C09130=1221.098,210.691,-57.647,-177.348,6.190,148.329
C09131=1221.102,210.442,-57.622,-177.351,6.188,148.329
C09132=1221.107,210.193,-57.597,-177.354,6.186,148.330
C09133=1221.111,209.944,-57.573,-177.356,6.184,148.330
C09134=1221.117,209.695,-57.549,-177.359,6.183,148.330
C09135=1221.121,209.446,-57.525,-177.361,6.181,148.331
C09136=1221.125,209.197,-57.501,-177.364,6.179,148.331
C09137=1221.130,208.949,-57.476,-177.367,6.177,148.331
C09138=1221.134,208.700,-57.452,-177.369,6.176,148.332
C09139=1221.138,208.451,-57.428,-177.371,6.174,148.332
C09140=1221.144,208.202,-57.404,-177.374,6.172,148.332
C09141=1221.148,207.953,-57.380,-177.377,6.171,148.333
C09142=1221.153,207.705,-57.356,-177.380,6.169,148.333
C09143=1221.158,207.456,-57.331,-177.382,6.167,148.334
C09144=1221.161,207.207,-57.307,-177.385,6.165,148.334
C09145=1221.166,206.958,-57.283,-177.388,6.163,148.334
C09146=1221.171,206.710,-57.259,-177.390,6.162,148.335
C09147=1221.176,206.461,-57.234,-177.392,6.161,148.335
C09148=1221.180,206.212,-57.211,-177.395,6.159,148.335
C09149=1221.185,205.964,-57.187,-177.398,6.157,148.336
C09150=1221.189,205.715,-57.163,-177.400,6.155,148.336
C09151=1221.194,205.466,-57.138,-177.403,6.153,148.336
C09152=1221.198,205.217,-57.115,-177.406,6.151,148.337
C09153=1221.203,204.968,-57.090,-177.408,6.150,148.337
C09154=1221.207,204.720,-57.066,-177.410,6.148,148.337
C09155=1221.213,204.471,-57.042,-177.413,6.147,148.338
C09156=1221.216,204.221,-57.018,-177.416,6.145,148.338
C09157=1221.221,203.973,-56.994,-177.418,6.143,148.338
C09158=1221.225,203.724,-56.971,-177.421,6.141,148.339
C09159=1221.230,203.476,-56.946,-177.424,6.139,148.339
C09160=1221.235,203.226,-56.923,-177.426,6.138,148.339
C09161=1221.240,202.978,-56.898,-177.428,6.136,148.340
C09162=1221.244,202.729,-56.875,-177.431,6.135,148.340
C09163=1221.248,202.480,-56.851,-177.434,6.133,148.340
C09164=1221.253,202.231,-56.827,-177.436,6.131,148.341
C09165=1221.257,201.982,-56.803,-177.439,6.129,148.341
C09166=1221.262,201.734,-56.779,-177.441,6.128,148.342
C09167=1221.267,201.485,-56.755,-177.444,6.126,148.342
C09168=1221.272,201.236,-56.731,-177.447,6.125,148.342
C09169=1221.276,200.987,-56.708,-177.449,6.123,148.343
C09170=1221.281,200.739,-56.684,-177.452,6.121,148.343
C09171=1221.285,200.490,-56.660,-177.454,6.120,148.344
C09172=1221.290,200.241,-56.636,-177.457,6.118,148.344
C09173=1221.294,199.992,-56.613,-177.459,6.116,148.344
C09174=1221.298,199.743,-56.588,-177.462,6.114,148.345
C09175=1221.303,199.494,-56.565,-177.465,6.113,148.345
C09176=1221.308,199.245,-56.542,-177.467,6.111,148.345
C09177=1221.312,198.997,-56.518,-177.469,6.110,148.346
C09178=1221.317,198.747,-56.494,-177.472,6.108,148.346
C09179=1221.322,198.499,-56.470,-177.475,6.106,148.347
C09180=1221.327,198.250,-56.446,-177.478,6.104,148.347
C09181=1221.331,198.001,-56.423,-177.480,6.103,148.347
C09182=1221.336,197.752,-56.399,-177.482,6.102,148.348
C09183=1221.340,197.503,-56.375,-177.485,6.100,148.348
C09184=1221.345,197.254,-56.352,-177.488,6.098,148.348
C09185=1221.349,197.006,-56.328,-177.490,6.096,148.349
C09186=1221.354,196.757,-56.305,-177.493,6.094,148.349
C09187=1221.359,196.508,-56.281,-177.495,6.093,148.349
C09188=1221.363,196.259,-56.257,-177.498,6.091,148.350
C09189=1221.368,196.010,-56.234,-177.500,6.090,148.350
C09190=1221.373,195.761,-56.211,-177.504,6.088,148.351
C09191=1221.377,195.512,-56.187,-177.506,6.086,148.351
C09192=1221.382,195.264,-56.163,-177.508,6.085,148.351
C09193=1221.386,195.015,-56.140,-177.511,6.083,148.352
C09194=1221.390,194.766,-56.117,-177.514,6.082,148.352
C09195=1221.395,194.517,-56.094,-177.516,6.080,148.352
C09196=1221.399,194.269,-56.070,-177.519,6.078,148.353
C09197=1221.404,194.020,-56.046,-177.521,6.077,148.353
C09198=1221.409,193.771,-56.023,-177.524,6.075,148.353
C09199=1221.414,193.522,-55.999,-177.526,6.073,148.354
C09200=1221.418,193.273,-55.976,-177.529,6.072,148.354
C09201=1221.423,193.024,-55.952,-177.531,6.071,148.355
C09202=1221.427,192.775,-55.929,-177.534,6.069,148.355
C09203=1221.433,192.527,-55.906,-177.537,6.067,148.355
C09204=1221.437,192.278,-55.883,-177.539,6.065,148.356
C09205=1221.441,192.029,-55.860,-177.541,6.064,148.356
C09206=1221.446,191.780,-55.836,-177.544,6.062,148.356
C09207=1221.451,191.531,-55.813,-177.547,6.060,148.357
C09208=1221.455,191.282,-55.789,-177.550,6.059,148.357
C09209=1221.460,191.033,-55.766,-177.553,6.057,148.358
C09210=1221.465,190.784,-55.743,-177.555,6.056,148.358
C09211=1221.468,190.536,-55.719,-177.557,6.054,148.358
C09212=1221.473,190.287,-55.696,-177.560,6.052,148.359
C09213=1221.478,190.038,-55.673,-177.563,6.051,148.359
C09214=1221.483,189.789,-55.650,-177.565,6.050,148.360
C09215=1221.488,189.540,-55.626,-177.567,6.048,148.360
C09216=1221.492,189.292,-55.603,-177.570,6.046,148.360
C09217=1221.497,189.043,-55.580,-177.573,6.044,148.361
C09218=1221.501,188.794,-55.557,-177.575,6.043,148.361
C09219=1221.506,188.545,-55.533,-177.578,6.042,148.362
C09220=1221.510,188.296,-55.511,-177.580,6.040,148.362
C09221=1221.515,188.047,-55.487,-177.583,6.038,148.362
C09222=1221.520,187.798,-55.465,-177.586,6.037,148.363
C09223=1221.525,187.549,-55.442,-177.588,6.035,148.363
C09224=1221.529,187.300,-55.419,-177.591,6.034,148.364
C09225=1221.534,187.051,-55.395,-177.593,6.033,148.364
C09226=1221.538,186.802,-55.372,-177.596,6.031,148.364
C09227=1221.543,186.553,-55.349,-177.598,6.029,148.365
C09228=1221.548,186.305,-55.326,-177.601,6.027,148.365
C09229=1221.552,186.056,-55.303,-177.604,6.026,148.366
C09230=1221.558,185.786,-55.278,-177.606,6.024,148.366
C09231=1221.562,185.517,-55.254,-177.609,6.023,148.366
C09232=1221.567,185.247,-55.229,-177.612,6.021,148.367
C09233=1221.572,184.977,-55.204,-177.615,6.019,148.367
C09234=1221.577,184.728,-55.181,-177.617,6.017,148.368
C09235=1221.581,184.479,-55.157,-177.620,6.016,148.368
C09236=1221.586,184.230,-55.135,-177.622,6.015,148.368
C09237=1221.590,183.981,-55.112,-177.625,6.013,148.369
C09238=1221.596,183.733,-55.089,-177.628,6.011,148.369
C09239=1221.600,183.484,-55.066,-177.631,6.009,148.370
C09240=1221.604,183.235,-55.043,-177.633,6.008,148.370
C09241=1221.609,182.985,-55.020,-177.635,6.007,148.370
C09242=1221.613,182.737,-54.997,-177.638,6.005,148.371
C09243=1221.619,182.488,-54.974,-177.640,6.004,148.371
C09244=1221.623,182.239,-54.952,-177.643,6.002,148.372
C09245=1221.628,181.990,-54.929,-177.646,6.000,148.372
C09246=1221.632,181.741,-54.906,-177.648,5.999,148.372
C09247=1221.637,181.493,-54.883,-177.651,5.998,148.373
C09248=1221.642,181.243,-54.861,-177.654,5.996,148.373
C09249=1221.646,180.994,-54.838,-177.656,5.994,148.374
C09250=1221.651,180.745,-54.815,-177.658,5.993,148.374
C09251=1221.655,180.497,-54.793,-177.661,5.991,148.374
C09252=1221.660,180.248,-54.769,-177.664,5.990,148.375
C09253=1221.664,179.998,-54.747,-177.666,5.989,148.375
C09254=1221.670,179.750,-54.724,-177.669,5.987,148.376
C09255=1221.674,179.501,-54.702,-177.672,5.985,148.376
C09256=1221.679,179.252,-54.679,-177.674,5.984,148.376
C09257=1221.683,179.003,-54.656,-177.676,5.982,148.377
C09258=1221.688,178.754,-54.634,-177.679,5.981,148.377
C09259=1221.692,178.505,-54.611,-177.682,5.980,148.378
C09260=1221.697,178.256,-54.589,-177.684,5.978,148.378
C09261=1221.702,178.008,-54.566,-177.687,5.976,148.378
C09262=1221.706,177.759,-54.543,-177.689,5.975,148.379
C09263=1221.711,177.509,-54.521,-177.692,5.974,148.379
C09264=1221.715,177.261,-54.498,-177.695,5.972,148.380
C09265=1221.720,177.012,-54.476,-177.697,5.971,148.380
C09266=1221.724,176.763,-54.453,-177.699,5.969,148.381
C09267=1221.730,176.514,-54.431,-177.703,5.968,148.381
C09268=1221.734,176.265,-54.409,-177.705,5.967,148.381
C09269=1221.739,176.016,-54.385,-177.707,5.965,148.382
C09270=1221.744,175.767,-54.364,-177.710,5.963,148.382
C09271=1221.748,175.518,-54.341,-177.712,5.962,148.383
C09272=1221.753,175.269,-54.318,-177.715,5.961,148.383
C09273=1221.757,175.021,-54.296,-177.718,5.959,148.384
C09274=1221.762,174.771,-54.273,-177.720,5.958,148.384
C09275=1221.767,174.522,-54.251,-177.723,5.956,148.384
C09276=1221.771,174.274,-54.229,-177.726,5.954,148.385
C09277=1221.776,174.024,-54.206,-177.728,5.953,148.385
C09278=1221.781,173.776,-54.184,-177.731,5.952,148.386
C09279=1221.785,173.526,-54.162,-177.733,5.950,148.386
C09280=1221.790,173.277,-54.139,-177.736,5.949,148.387
C09281=1221.794,173.029,-54.117,-177.738,5.947,148.387
C09282=1221.799,172.779,-54.095,-177.741,5.945,148.387
C09283=1221.804,172.531,-54.072,-177.743,5.944,148.388
C09284=1221.809,172.281,-54.050,-177.746,5.943,148.388
C09285=1221.813,172.033,-54.028,-177.748,5.942,148.389
C09286=1221.818,171.784,-54.005,-177.751,5.940,148.389
C09287=1221.822,171.534,-53.983,-177.754,5.938,148.389
C09288=1221.827,171.286,-53.961,-177.756,5.938,148.390
C09289=1221.831,171.037,-53.939,-177.759,5.936,148.390
C09290=1221.837,170.788,-53.916,-177.762,5.934,148.391
C09291=1221.841,170.539,-53.894,-177.764,5.933,148.391
C09292=1221.846,170.291,-53.872,-177.767,5.931,148.392
C09293=1221.851,170.041,-53.849,-177.770,5.930,148.392
C09294=1221.856,169.792,-53.828,-177.772,5.929,148.392
C09295=1221.860,169.543,-53.806,-177.774,5.927,148.393
C09296=1221.864,169.294,-53.784,-177.777,5.926,148.393
C09297=1221.869,169.045,-53.762,-177.780,5.924,148.394
C09298=1221.874,168.796,-53.738,-177.782,5.923,148.394
C09299=1221.879,168.547,-53.717,-177.784,5.922,148.394
C09300=1221.883,168.298,-53.695,-177.787,5.920,148.395
C09301=1221.888,168.049,-53.673,-177.790,5.919,148.395
C09302=1221.893,167.800,-53.650,-177.792,5.917,148.396
C09303=1221.898,167.551,-53.629,-177.795,5.915,148.396
C09304=1221.902,167.302,-53.607,-177.797,5.915,148.397
C09305=1221.907,167.053,-53.585,-177.800,5.913,148.397
C09306=1221.911,166.804,-53.562,-177.803,5.911,148.398
C09307=1221.916,166.556,-53.541,-177.805,5.910,148.398
C09308=1221.920,166.306,-53.518,-177.808,5.909,148.399
C09309=1221.925,166.057,-53.496,-177.810,5.908,148.399
C09310=1221.930,165.808,-53.474,-177.813,5.906,148.399
C09311=1221.935,165.559,-53.452,-177.815,5.905,148.400
C09312=1221.939,165.310,-53.430,-177.818,5.903,148.400
C09313=1221.944,165.061,-53.409,-177.821,5.901,148.401
C09314=1221.949,164.813,-53.387,-177.823,5.901,148.401
C09315=1221.953,164.563,-53.365,-177.826,5.899,148.402
C09316=1221.958,164.315,-53.343,-177.828,5.898,148.402
C09317=1221.962,164.065,-53.321,-177.831,5.896,148.402
C09318=1221.968,163.816,-53.299,-177.834,5.895,148.403
C09319=1221.972,163.567,-53.277,-177.836,5.894,148.403
C09320=1221.977,163.318,-53.255,-177.839,5.892,148.404
C09321=1221.981,163.069,-53.233,-177.841,5.891,148.404
C09322=1221.986,162.820,-53.212,-177.844,5.889,148.405
C09323=1221.991,162.571,-53.191,-177.847,5.888,148.405
C09324=1221.995,162.322,-53.169,-177.849,5.887,148.406
C09325=1222.000,162.073,-53.147,-177.852,5.885,148.406
C09326=1222.004,161.824,-53.125,-177.854,5.884,148.406
C09327=1222.009,161.575,-53.103,-177.857,5.883,148.407
C09328=1222.014,161.327,-53.081,-177.859,5.882,148.407
C09329=1222.018,161.077,-53.059,-177.862,5.880,148.408
C09330=1222.024,160.828,-53.038,-177.864,5.878,148.408
C09331=1222.028,160.579,-53.016,-177.867,5.877,148.409
C09332=1222.033,160.330,-52.995,-177.870,5.876,148.409
C09333=1222.038,160.081,-52.973,-177.872,5.875,148.410
C09334=1222.042,159.812,-52.950,-177.875,5.873,148.410
C09335=1222.048,159.544,-52.926,-177.878,5.871,148.410
C09336=1222.052,159.274,-52.902,-177.881,5.870,148.411
C09337=1222.057,159.004,-52.880,-177.883,5.869,148.411
C09338=1222.062,158.756,-52.858,-177.886,5.867,148.412
C09339=1222.067,158.507,-52.836,-177.888,5.866,148.412
C09340=1222.071,158.257,-52.815,-177.891,5.865,148.413
C09341=1222.076,158.009,-52.793,-177.893,5.864,148.413
C09342=1222.081,157.760,-52.772,-177.896,5.862,148.414
C09343=1222.085,157.511,-52.750,-177.899,5.860,148.414
C09344=1222.091,157.261,-52.729,-177.901,5.860,148.415
C09345=1222.096,157.013,-52.707,-177.904,5.858,148.415
C09346=1222.099,156.764,-52.685,-177.906,5.857,148.416
C09347=1222.104,156.514,-52.665,-177.909,5.855,148.416
C09348=1222.109,156.266,-52.643,-177.911,5.854,148.417
C09349=1222.113,156.016,-52.621,-177.914,5.853,148.417
C09350=1222.119,155.767,-52.600,-177.917,5.852,148.418
C09351=1222.123,155.519,-52.578,-177.919,5.850,148.418
C09352=1222.128,155.270,-52.556,-177.922,5.849,148.419
C09353=1222.133,155.020,-52.535,-177.924,5.848,148.419
C09354=1222.137,154.772,-52.514,-177.927,5.847,148.419
C09355=1222.142,154.522,-52.493,-177.930,5.845,148.420
C09356=1222.146,154.273,-52.471,-177.932,5.843,148.420
C09357=1222.152,154.024,-52.450,-177.934,5.842,148.421
C09358=1222.156,153.775,-52.428,-177.938,5.841,148.421
C09359=1222.161,153.527,-52.407,-177.940,5.840,148.422
C09360=1222.165,153.277,-52.386,-177.942,5.838,148.422
C09361=1222.170,153.028,-52.364,-177.945,5.837,148.423
C09362=1222.175,152.779,-52.343,-177.948,5.836,148.423
C09363=1222.180,152.530,-52.322,-177.950,5.835,148.423
C09364=1222.184,152.281,-52.301,-177.953,5.833,148.424
C09365=1222.189,152.032,-52.279,-177.955,5.832,148.424
C09366=1222.194,151.783,-52.258,-177.958,5.831,148.425
C09367=1222.199,151.534,-52.237,-177.960,5.830,148.425
C09368=1222.203,151.285,-52.216,-177.963,5.828,148.426
C09369=1222.208,151.036,-52.194,-177.966,5.827,148.426
C09370=1222.213,150.787,-52.173,-177.968,5.825,148.427
C09371=1222.218,150.537,-52.152,-177.970,5.824,148.427
C09372=1222.222,150.289,-52.131,-177.973,5.823,148.428
C09373=1222.227,150.039,-52.110,-177.976,5.822,148.428
C09374=1222.231,149.790,-52.088,-177.979,5.820,148.429
C09375=1222.236,149.541,-52.068,-177.981,5.820,148.429
C09376=1222.241,149.292,-52.047,-177.984,5.818,148.430
C09377=1222.246,149.044,-52.025,-177.986,5.817,148.430
C09378=1222.250,148.794,-52.004,-177.989,5.815,148.431
C09379=1222.255,148.545,-51.983,-177.991,5.814,148.431
C09380=1222.260,148.296,-51.962,-177.994,5.813,148.432
C09381=1222.264,148.047,-51.941,-177.996,5.812,148.432
C09382=1222.269,147.798,-51.920,-177.999,5.810,148.433
C09383=1222.274,147.549,-51.899,-178.001,5.809,148.433
C09384=1222.278,147.299,-51.878,-178.004,5.808,148.433
C09385=1222.283,147.050,-51.857,-178.007,5.807,148.434
C09386=1222.288,146.802,-51.835,-178.009,5.805,148.434
C09387=1222.293,146.553,-51.815,-178.012,5.804,148.435
C09388=1222.298,146.303,-51.794,-178.015,5.803,148.435
C09389=1222.302,146.054,-51.774,-178.017,5.802,148.436
C09390=1222.307,145.806,-51.752,-178.019,5.801,148.436
C09391=1222.312,145.556,-51.731,-178.022,5.799,148.437
C09392=1222.316,145.307,-51.710,-178.025,5.799,148.437
C09393=1222.321,145.058,-51.689,-178.027,5.797,148.438
C09394=1222.325,144.809,-51.668,-178.029,5.796,148.438
C09395=1222.331,144.560,-51.647,-178.033,5.794,148.439
C09396=1222.335,144.311,-51.627,-178.035,5.793,148.439
C09397=1222.340,144.062,-51.606,-178.038,5.792,148.440
C09398=1222.345,143.813,-51.585,-178.040,5.791,148.440
C09399=1222.349,143.563,-51.564,-178.043,5.789,148.441
C09400=1222.354,143.314,-51.542,-178.045,5.788,148.441
C09401=1222.359,143.065,-51.522,-178.048,5.787,148.441
C09402=1222.364,142.816,-51.501,-178.050,5.786,148.442
C09403=1222.368,142.567,-51.481,-178.053,5.785,148.443
C09404=1222.373,142.318,-51.460,-178.056,5.784,148.443
C09405=1222.378,142.069,-51.439,-178.058,5.783,148.444
C09406=1222.383,141.820,-51.418,-178.061,5.781,148.444
C09407=1222.387,141.571,-51.398,-178.063,5.780,148.445
C09408=1222.392,141.322,-51.378,-178.066,5.778,148.445
C09409=1222.397,141.073,-51.356,-178.068,5.778,148.446
C09410=1222.401,140.824,-51.336,-178.071,5.776,148.446
C09411=1222.406,140.575,-51.315,-178.074,5.775,148.447
C09412=1222.411,140.326,-51.294,-178.076,5.774,148.447
C09413=1222.416,140.077,-51.273,-178.079,5.773,148.448
C09414=1222.420,139.827,-51.253,-178.081,5.772,148.448
C09415=1222.425,139.578,-51.232,-178.084,5.770,148.448
C09416=1222.429,139.329,-51.211,-178.086,5.769,148.449
C09417=1222.434,139.080,-51.191,-178.089,5.768,148.449
C09418=1222.439,138.831,-51.170,-178.092,5.767,148.450
C09419=1222.443,138.582,-51.150,-178.094,5.765,148.450
C09420=1222.449,138.332,-51.129,-178.097,5.764,148.451
C09421=1222.453,138.083,-51.108,-178.099,5.764,148.451
C09422=1222.458,137.834,-51.089,-178.102,5.762,148.452
C09423=1222.463,137.585,-51.068,-178.104,5.761,148.452
C09424=1222.467,137.336,-51.047,-178.107,5.759,148.453
C09425=1222.473,137.086,-51.026,-178.109,5.759,148.453
C09426=1222.477,136.837,-51.006,-178.112,5.758,148.454
C09427=1222.481,136.588,-50.985,-178.115,5.756,148.454
C09428=1222.487,136.339,-50.965,-178.117,5.755,148.455
C09429=1222.491,136.090,-50.944,-178.120,5.754,148.455
C09430=1222.495,135.841,-50.924,-178.122,5.753,148.456
C09431=1222.502,135.592,-50.904,-178.125,5.751,148.456
C09432=1222.506,135.343,-50.884,-178.127,5.750,148.457
C09433=1222.510,135.094,-50.863,-178.130,5.750,148.457
C09434=1222.516,134.845,-50.842,-178.133,5.748,148.458
C09435=1222.520,134.596,-50.822,-178.135,5.747,148.459
C09436=1222.524,134.347,-50.801,-178.138,5.745,148.459
C09437=1222.529,134.098,-50.782,-178.140,5.745,148.459
C09438=1222.535,133.829,-50.759,-178.143,5.743,148.460
C09439=1222.540,133.560,-50.737,-178.146,5.742,148.461
C09440=1222.544,133.291,-50.716,-178.149,5.741,148.461
C09441=1222.550,133.023,-50.694,-178.151,5.740,148.462
C09442=1222.554,132.774,-50.673,-178.154,5.739,148.462
C09443=1222.559,132.524,-50.653,-178.156,5.738,148.463
C09444=1222.564,132.275,-50.632,-178.159,5.737,148.463
C09445=1222.569,132.026,-50.612,-178.162,5.735,148.464
C09446=1222.574,131.778,-50.592,-178.164,5.734,148.464
C09447=1222.578,131.529,-50.572,-178.167,5.733,148.465
C09448=1222.584,131.279,-50.552,-178.170,5.732,148.465
C09449=1222.588,131.030,-50.531,-178.172,5.731,148.466
C09450=1222.592,130.781,-50.511,-178.174,5.729,148.466
C09451=1222.597,130.531,-50.491,-178.177,5.729,148.467
C09452=1222.602,130.282,-50.471,-178.180,5.727,148.467
C09453=1222.607,130.033,-50.450,-178.182,5.726,148.468
C09454=1222.612,129.783,-50.430,-178.184,5.725,148.468
C09455=1222.617,129.535,-50.410,-178.188,5.724,148.469
C09456=1222.621,129.286,-50.390,-178.190,5.723,148.469
C09457=1222.626,129.037,-50.370,-178.192,5.722,148.470
C09458=1222.630,128.788,-50.350,-178.195,5.720,148.470
C09459=1222.636,128.538,-50.330,-178.198,5.720,148.471
C09460=1222.640,128.289,-50.309,-178.200,5.718,148.471
C09461=1222.645,128.040,-50.289,-178.203,5.717,148.472
C09462=1222.650,127.791,-50.270,-178.205,5.716,148.472
C09463=1222.654,127.542,-50.249,-178.208,5.715,148.473
C09464=1222.659,127.293,-50.230,-178.210,5.714,148.473
C09465=1222.664,127.044,-50.209,-178.213,5.713,148.474
C09466=1222.668,126.794,-50.190,-178.216,5.712,148.474
C09467=1222.673,126.546,-50.170,-178.218,5.711,148.475
C09468=1222.679,126.296,-50.149,-178.221,5.710,148.476
C09469=1222.683,126.047,-50.129,-178.223,5.708,148.476
C09470=1222.688,125.797,-50.109,-178.226,5.708,148.477
C09471=1222.692,125.549,-50.089,-178.229,5.706,148.477
C09472=1222.697,125.299,-50.069,-178.231,5.705,148.478
C09473=1222.702,125.051,-50.049,-178.233,5.704,148.478
C09474=1222.707,124.801,-50.030,-178.237,5.703,148.479
C09475=1222.712,124.552,-50.010,-178.239,5.702,148.479
C09476=1222.716,124.303,-49.990,-178.241,5.701,148.480
C09477=1222.721,124.054,-49.970,-178.244,5.700,148.480
C09478=1222.726,123.805,-49.950,-178.247,5.699,148.481
C09479=1222.731,123.555,-49.930,-178.249,5.698,148.481
C09480=1222.735,123.306,-49.911,-178.252,5.697,148.482
C09481=1222.740,123.057,-49.890,-178.254,5.696,148.482
C09482=1222.745,122.808,-49.871,-178.257,5.695,148.483
C09483=1222.750,122.558,-49.851,-178.259,5.693,148.483
C09484=1222.754,122.309,-49.831,-178.262,5.693,148.484
C09485=1222.759,122.060,-49.811,-178.264,5.692,148.484
C09486=1222.764,121.812,-49.791,-178.267,5.690,148.485
C09487=1222.769,121.562,-49.772,-178.270,5.690,148.485
C09488=1222.774,121.312,-49.752,-178.272,5.689,148.486
C09489=1222.779,121.064,-49.733,-178.275,5.687,148.486
C09490=1222.783,120.815,-49.712,-178.277,5.686,148.487
C09491=1222.788,120.565,-49.693,-178.280,5.686,148.487
C09492=1222.792,120.316,-49.674,-178.282,5.684,148.488
C09493=1222.797,120.067,-49.654,-178.285,5.683,148.489
C09494=1222.802,119.818,-49.634,-178.287,5.682,148.489
C09495=1222.807,119.568,-49.614,-178.290,5.681,148.490
C09496=1222.812,119.319,-49.595,-178.292,5.680,148.490
C09497=1222.817,119.070,-49.575,-178.295,5.679,148.491
C09498=1222.821,118.821,-49.555,-178.298,5.679,148.491
C09499=1222.827,118.572,-49.536,-178.300,5.677,148.492
C09500=1222.831,118.323,-49.516,-178.303,5.676,148.492
C09501=1222.836,118.073,-49.496,-178.305,5.675,148.493
C09502=1222.841,117.824,-49.478,-178.308,5.674,148.493
C09503=1222.845,117.575,-49.457,-178.310,5.673,148.494
C09504=1222.850,117.326,-49.438,-178.313,5.672,148.494
C09505=1222.855,117.077,-49.418,-178.316,5.671,148.495
C09506=1222.860,116.827,-49.399,-178.318,5.670,148.495
C09507=1222.865,116.578,-49.379,-178.321,5.669,148.496
C09508=1222.869,116.329,-49.360,-178.324,5.667,148.496
C09509=1222.874,116.080,-49.341,-178.326,5.667,148.497
C09510=1222.878,115.831,-49.320,-178.328,5.666,148.497
C09511=1222.884,115.582,-49.301,-178.331,5.665,148.498
C09512=1222.889,115.332,-49.281,-178.334,5.663,148.499
C09513=1222.893,115.083,-49.262,-178.336,5.663,148.499
C09514=1222.898,114.834,-49.243,-178.339,5.662,148.500
C09515=1222.903,114.585,-49.223,-178.342,5.660,148.500
C09516=1222.908,114.336,-49.204,-178.344,5.660,148.501
C09517=1222.913,114.086,-49.184,-178.346,5.659,148.501
C09518=1222.917,113.837,-49.165,-178.349,5.658,148.502
C09519=1222.922,113.588,-49.146,-178.352,5.657,148.503
C09520=1222.927,113.339,-49.126,-178.354,5.656,148.503
C09521=1222.932,113.090,-49.107,-178.357,5.655,148.504
C09522=1222.936,112.840,-49.088,-178.359,5.653,148.504
C09523=1222.941,112.591,-49.068,-178.362,5.653,148.505
C09524=1222.946,112.342,-49.049,-178.364,5.652,148.505
C09525=1222.951,112.092,-49.030,-178.367,5.651,148.506
C09526=1222.956,111.844,-49.011,-178.370,5.650,148.506
C09527=1222.960,111.594,-48.991,-178.372,5.649,148.507
C09528=1222.966,111.345,-48.972,-178.375,5.648,148.507
C09529=1222.970,111.096,-48.953,-178.377,5.647,148.508
C09530=1222.974,110.847,-48.933,-178.380,5.646,148.508
C09531=1222.980,110.598,-48.914,-178.383,5.645,148.509
C09532=1222.984,110.348,-48.896,-178.385,5.644,148.509
C09533=1222.989,110.099,-48.876,-178.387,5.644,148.510
C09534=1222.994,109.849,-48.857,-178.390,5.642,148.510
C09535=1222.999,109.601,-48.838,-178.393,5.641,148.511
C09536=1223.004,109.351,-48.818,-178.395,5.640,148.512
C09537=1223.009,109.102,-48.799,-178.398,5.639,148.512
C09538=1223.013,108.853,-48.780,-178.401,5.638,148.513
C09539=1223.019,108.604,-48.761,-178.403,5.637,148.513
C09540=1223.023,108.354,-48.742,-178.405,5.637,148.514
C09541=1223.028,108.106,-48.723,-178.409,5.635,148.514
C09542=1223.033,107.837,-48.702,-178.411,5.634,148.515
C09543=1223.038,107.568,-48.681,-178.413,5.634,148.516
C09544=1223.044,107.300,-48.661,-178.416,5.632,148.516
C09545=1223.048,107.031,-48.640,-178.419,5.631,148.517
C09546=1223.053,106.783,-48.621,-178.422,5.631,148.517
C09547=1223.059,106.533,-48.602,-178.424,5.629,148.518
C09548=1223.063,106.284,-48.583,-178.427,5.628,148.519
C09549=1223.068,106.035,-48.564,-178.429,5.628,148.519
C09550=1223.072,105.786,-48.545,-178.432,5.627,148.520
C09551=1223.078,105.536,-48.526,-178.435,5.625,148.520
C09552=1223.082,105.287,-48.507,-178.437,5.625,148.521
C09553=1223.087,105.038,-48.488,-178.440,5.624,148.521
C09554=1223.091,104.788,-48.470,-178.442,5.623,148.522
C09555=1223.097,104.539,-48.450,-178.445,5.622,148.522
C09556=1223.101,104.290,-48.431,-178.448,5.621,148.523
C09557=1223.106,104.041,-48.413,-178.450,5.620,148.523
C09558=1223.111,103.791,-48.393,-178.452,5.619,148.524
C09559=1223.116,103.542,-48.374,-178.455,5.618,148.525
C09560=1223.121,103.293,-48.356,-178.458,5.617,148.525
C09561=1223.125,103.044,-48.337,-178.460,5.616,148.526
C09562=1223.131,102.795,-48.318,-178.463,5.616,148.526
C09563=1223.135,102.545,-48.299,-178.465,5.615,148.527
C09564=1223.140,102.296,-48.280,-178.468,5.613,148.527
C09565=1223.145,102.046,-48.262,-178.471,5.613,148.528
C09566=1223.149,101.798,-48.243,-178.473,5.612,148.528
C09567=1223.155,101.549,-48.224,-178.475,5.611,148.529
C09568=1223.159,101.299,-48.205,-178.478,5.609,148.530
C09569=1223.164,101.050,-48.186,-178.481,5.609,148.530
C09570=1223.169,100.800,-48.168,-178.483,5.608,148.531
C09571=1223.174,100.551,-48.148,-178.486,5.607,148.531
C09572=1223.179,100.302,-48.130,-178.488,5.607,148.532
C09573=1223.183,100.053,-48.111,-178.491,5.605,148.533
C09574=1223.188,99.803,-48.093,-178.493,5.604,148.533
C09575=1223.192,99.554,-48.074,-178.496,5.604,148.534
C09576=1223.198,99.305,-48.055,-178.499,5.603,148.534
C09577=1223.203,99.056,-48.036,-178.501,5.602,148.535
C09578=1223.207,98.806,-48.018,-178.504,5.601,148.535
C09579=1223.212,98.557,-47.999,-178.507,5.600,148.536
C09580=1223.217,98.308,-47.981,-178.509,5.599,148.536
C09581=1223.221,98.059,-47.962,-178.511,5.599,148.537
C09582=1223.227,97.809,-47.943,-178.514,5.598,148.538
C09583=1223.232,97.561,-47.924,-178.517,5.596,148.538
C09584=1223.237,97.311,-47.905,-178.519,5.596,148.539
C09585=1223.242,97.061,-47.887,-178.522,5.595,148.539
C09586=1223.246,96.813,-47.869,-178.524,5.594,148.540
C09587=1223.251,96.563,-47.850,-178.527,5.593,148.540
C09588=1223.256,96.314,-47.831,-178.529,5.593,148.541
C09589=1223.261,96.065,-47.813,-178.532,5.591,148.541
C09590=1223.265,95.815,-47.795,-178.535,5.590,148.542
C09591=1223.270,95.566,-47.776,-178.537,5.590,148.543
C09592=1223.275,95.317,-47.758,-178.539,5.589,148.543
C09593=1223.280,95.067,-47.739,-178.542,5.588,148.544
C09594=1223.285,94.818,-47.720,-178.545,5.587,148.544
C09595=1223.290,94.569,-47.702,-178.547,5.586,148.545
C09596=1223.294,94.319,-47.684,-178.550,5.585,148.546
C09597=1223.299,94.071,-47.665,-178.553,5.585,148.546
C09598=1223.304,93.821,-47.646,-178.555,5.584,148.547
C09599=1223.309,93.572,-47.628,-178.557,5.583,148.547
C09600=1223.313,93.323,-47.609,-178.560,5.582,148.548
C09601=1223.318,93.074,-47.591,-178.563,5.581,148.548
C09602=1223.324,92.824,-47.573,-178.565,5.580,148.549
C09603=1223.328,92.574,-47.554,-178.568,5.580,148.550
C09604=1223.333,92.326,-47.536,-178.570,5.579,148.550
C09605=1223.338,92.077,-47.518,-178.573,5.578,148.551
C09606=1223.343,91.827,-47.499,-178.576,5.577,148.551
C09607=1223.348,91.577,-47.481,-178.578,5.576,148.552
C09608=1223.352,91.329,-47.462,-178.581,5.575,148.552
C09609=1223.357,91.079,-47.444,-178.583,5.574,148.553
C09610=1223.362,90.830,-47.426,-178.586,5.574,148.554
C09611=1223.366,90.580,-47.408,-178.588,5.573,148.554
C09612=1223.372,90.331,-47.389,-178.591,5.571,148.555
C09613=1223.377,90.082,-47.371,-178.594,5.571,148.555
C09614=1223.382,89.833,-47.353,-178.596,5.570,148.556
C09615=1223.386,89.584,-47.335,-178.598,5.569,148.557
C09616=1223.391,89.334,-47.316,-178.601,5.569,148.557
C09617=1223.396,89.085,-47.298,-178.603,5.568,148.558
C09618=1223.401,88.835,-47.280,-178.606,5.567,148.558
C09619=1223.406,88.586,-47.262,-178.609,5.566,148.559
C09620=1223.411,88.337,-47.244,-178.612,5.565,148.560
C09621=1223.416,88.087,-47.225,-178.614,5.564,148.560
C09622=1223.420,87.839,-47.207,-178.616,5.564,148.561
C09623=1223.425,87.589,-47.189,-178.619,5.563,148.561
C09624=1223.430,87.340,-47.171,-178.621,5.562,148.562
C09625=1223.435,87.091,-47.153,-178.624,5.561,148.562
C09626=1223.439,86.841,-47.134,-178.627,5.560,148.563
C09627=1223.444,86.592,-47.116,-178.630,5.559,148.564
C09628=1223.450,86.343,-47.098,-178.632,5.559,148.564
C09629=1223.455,86.093,-47.080,-178.634,5.558,148.565
C09630=1223.460,85.844,-47.062,-178.637,5.557,148.565
C09631=1223.464,85.595,-47.044,-178.639,5.556,148.566
C09632=1223.469,85.345,-47.026,-178.642,5.556,148.566
C09633=1223.474,85.096,-47.008,-178.645,5.554,148.567
C09634=1223.479,84.847,-46.990,-178.648,5.554,148.568
C09635=1223.483,84.598,-46.972,-178.650,5.553,148.568
C09636=1223.488,84.348,-46.954,-178.652,5.552,148.569
C09637=1223.493,84.099,-46.936,-178.655,5.552,148.570
C09638=1223.498,83.850,-46.918,-178.657,5.551,148.570
C09639=1223.503,83.601,-46.900,-178.660,5.550,148.571
C09640=1223.507,83.351,-46.881,-178.662,5.550,148.571
C09641=1223.513,83.101,-46.864,-178.665,5.549,148.572
C09642=1223.518,82.852,-46.846,-178.668,5.547,148.572
C09643=1223.522,82.603,-46.828,-178.670,5.547,148.573
C09644=1223.527,82.354,-46.810,-178.673,5.546,148.574
C09645=1223.532,82.105,-46.792,-178.675,5.545,148.574
C09646=1223.537,81.836,-46.773,-178.678,5.545,148.575
C09647=1223.542,81.568,-46.753,-178.680,5.544,148.575
C09648=1223.548,81.299,-46.735,-178.683,5.542,148.576
C09649=1223.553,81.031,-46.715,-178.686,5.542,148.577
C09650=1223.558,80.782,-46.697,-178.689,5.541,148.577
C09651=1223.563,80.533,-46.679,-178.691,5.541,148.578
C09652=1223.568,80.283,-46.661,-178.694,5.540,148.579
C09653=1223.573,80.034,-46.644,-178.696,5.539,148.579
C09654=1223.578,79.784,-46.626,-178.699,5.538,148.580
C09655=1223.583,79.535,-46.608,-178.702,5.537,148.580
C09656=1223.588,79.286,-46.590,-178.705,5.537,148.581
C09657=1223.592,79.037,-46.573,-178.707,5.536,148.581
C09658=1223.597,78.787,-46.555,-178.709,5.535,148.582
C09659=1223.601,78.538,-46.537,-178.712,5.534,148.583
C09660=1223.606,78.288,-46.519,-178.715,5.534,148.583
C09661=1223.611,78.039,-46.502,-178.717,5.533,148.584
C09662=1223.616,77.789,-46.484,-178.719,5.532,148.584
C09663=1223.621,77.540,-46.466,-178.722,5.532,148.585
C09664=1223.625,77.291,-46.448,-178.725,5.531,148.586
C09665=1223.631,77.042,-46.431,-178.727,5.529,148.586
C09666=1223.636,76.792,-46.413,-178.730,5.529,148.587
C09667=1223.641,76.543,-46.395,-178.732,5.528,148.588
C09668=1223.646,76.293,-46.378,-178.735,5.528,148.588
C09669=1223.651,76.044,-46.360,-178.737,5.527,148.589
C09670=1223.655,75.795,-46.343,-178.740,5.526,148.589
C09671=1223.660,75.546,-46.325,-178.743,5.526,148.590
C09672=1223.665,75.296,-46.307,-178.745,5.525,148.591
C09673=1223.670,75.047,-46.289,-178.747,5.524,148.591
C09674=1223.675,74.797,-46.272,-178.750,5.523,148.592
C09675=1223.679,74.549,-46.255,-178.753,5.523,148.592
C09676=1223.684,74.299,-46.237,-178.755,5.522,148.593
C09677=1223.689,74.050,-46.220,-178.757,5.521,148.593
C09678=1223.694,73.800,-46.202,-178.760,5.520,148.594
C09679=1223.700,73.551,-46.184,-178.763,5.519,148.595
C09680=1223.704,73.302,-46.167,-178.766,5.519,148.595
C09681=1223.709,73.052,-46.150,-178.768,5.518,148.596
C09682=1223.714,72.804,-46.132,-178.771,5.517,148.597
C09683=1223.719,72.555,-46.115,-178.773,5.517,148.597
C09684=1223.724,72.305,-46.097,-178.776,5.516,148.598
C09685=1223.729,72.056,-46.079,-178.778,5.516,148.598
C09686=1223.734,71.806,-46.062,-178.781,5.515,148.599
C09687=1223.738,71.557,-46.045,-178.783,5.514,148.600
C09688=1223.743,71.307,-46.027,-178.786,5.513,148.600
C09689=1223.748,71.058,-46.009,-178.788,5.513,148.601
C09690=1223.753,70.809,-45.993,-178.791,5.512,148.602
C09691=1223.758,70.559,-45.975,-178.793,5.511,148.602
C09692=1223.763,70.310,-45.958,-178.796,5.511,148.603
C09693=1223.768,70.060,-45.940,-178.798,5.510,148.603
C09694=1223.772,69.811,-45.923,-178.801,5.510,148.604
C09695=1223.777,69.561,-45.906,-178.803,5.509,148.604
C09696=1223.783,69.313,-45.888,-178.806,5.507,148.605
C09697=1223.787,69.063,-45.871,-178.809,5.507,148.606
C09698=1223.792,68.814,-45.853,-178.812,5.506,148.606
C09699=1223.797,68.565,-45.837,-178.814,5.506,148.607
C09700=1223.802,68.315,-45.819,-178.816,5.505,148.607
C09701=1223.807,68.066,-45.801,-178.819,5.504,148.608
C09702=1223.811,67.816,-45.785,-178.822,5.503,148.609
C09703=1223.816,67.567,-45.767,-178.824,5.503,148.609
C09704=1223.822,67.317,-45.750,-178.827,5.502,148.610
C09705=1223.827,67.068,-45.733,-178.829,5.501,148.611
C09706=1223.832,66.819,-45.715,-178.832,5.501,148.611
C09707=1223.836,66.570,-45.699,-178.834,5.500,148.612
C09708=1223.841,66.320,-45.681,-178.837,5.500,148.613
C09709=1223.845,66.071,-45.664,-178.840,5.499,148.613
C09710=1223.851,65.821,-45.647,-178.842,5.498,148.614
C09711=1223.856,65.571,-45.629,-178.844,5.498,148.614
C09712=1223.861,65.323,-45.612,-178.847,5.497,148.615
C09713=1223.866,65.073,-45.595,-178.850,5.496,148.616
C09714=1223.870,64.824,-45.578,-178.852,5.496,148.616
C09715=1223.875,64.575,-45.561,-178.854,5.495,148.617
C09716=1223.880,64.325,-45.544,-178.857,5.494,148.617
C09717=1223.885,64.075,-45.527,-178.860,5.494,148.618
C09718=1223.890,63.827,-45.510,-178.862,5.493,148.619
C09719=1223.895,63.578,-45.492,-178.865,5.493,148.619
C09720=1223.899,63.328,-45.476,-178.867,5.492,148.620
C09721=1223.905,63.078,-45.458,-178.870,5.491,148.620
C09722=1223.909,62.829,-45.442,-178.872,5.490,148.621
C09723=1223.915,62.580,-45.425,-178.875,5.490,148.622
C09724=1223.919,62.331,-45.407,-178.878,5.489,148.622
C09725=1223.924,62.081,-45.390,-178.880,5.488,148.623
C09726=1223.929,61.832,-45.373,-178.882,5.488,148.624
C09727=1223.934,61.582,-45.356,-178.885,5.487,148.624
C09728=1223.939,61.333,-45.340,-178.888,5.487,148.625
C09729=1223.944,61.083,-45.323,-178.890,5.486,148.626
C09730=1223.949,60.834,-45.305,-178.893,5.486,148.626
C09731=1223.954,60.585,-45.288,-178.895,5.485,148.627
C09732=1223.959,60.336,-45.272,-178.898,5.484,148.627
C09733=1223.964,60.086,-45.254,-178.900,5.483,148.628
C09734=1223.969,59.836,-45.238,-178.903,5.483,148.629
C09735=1223.973,59.587,-45.221,-178.906,5.482,148.629
C09736=1223.979,59.338,-45.204,-178.908,5.482,148.630
C09737=1223.983,59.088,-45.188,-178.910,5.481,148.630
C09738=1223.989,58.839,-45.170,-178.913,5.480,148.631
C09739=1223.993,58.589,-45.154,-178.916,5.480,148.632
C09740=1223.999,58.341,-45.136,-178.918,5.479,148.632
C09741=1224.003,58.091,-45.119,-178.921,5.479,148.633
C09742=1224.007,57.842,-45.103,-178.923,5.478,148.634
C09743=1224.013,57.593,-45.086,-178.926,5.477,148.634
C09744=1224.018,57.343,-45.069,-178.928,5.476,148.635
C09745=1224.022,57.094,-45.052,-178.931,5.476,148.636
C09746=1224.027,56.844,-45.035,-178.934,5.475,148.636
C09747=1224.033,56.595,-45.019,-178.936,5.475,148.637
C09748=1224.038,56.345,-45.002,-178.938,5.474,148.637
C09749=1224.042,56.096,-44.985,-178.941,5.473,148.638
C09750=1224.048,55.827,-44.968,-178.944,5.473,148.639
C09751=1224.053,55.558,-44.949,-178.946,5.472,148.639
C09752=1224.058,55.291,-44.931,-178.949,5.471,148.640
C09753=1224.063,55.022,-44.913,-178.953,5.471,148.641
C09754=1224.069,54.773,-44.896,-178.955,5.470,148.641
C09755=1224.073,54.523,-44.880,-178.957,5.469,148.642
C09756=1224.078,54.274,-44.863,-178.960,5.468,148.643
C09757=1224.084,54.025,-44.846,-178.963,5.468,148.643
C09758=1224.088,53.775,-44.830,-178.965,5.467,148.644
C09759=1224.093,53.525,-44.814,-178.968,5.467,148.645
C09760=1224.098,53.276,-44.797,-178.970,5.466,148.645
C09761=1224.103,53.027,-44.780,-178.973,5.465,148.646
C09762=1224.108,52.777,-44.763,-178.975,5.466,148.646
C09763=1224.113,52.528,-44.747,-178.977,5.465,148.647
C09764=1224.118,52.279,-44.730,-178.980,5.464,148.648
C09765=1224.123,52.029,-44.713,-178.983,5.464,148.648
C09766=1224.128,51.780,-44.698,-178.985,5.463,148.649
C09767=1224.132,51.530,-44.681,-178.987,5.462,148.650
C09768=1224.137,51.281,-44.665,-178.990,5.462,148.650
C09769=1224.143,51.032,-44.647,-178.993,5.461,148.651
C09770=1224.147,50.782,-44.631,-178.995,5.461,148.652
C09771=1224.153,50.533,-44.615,-178.998,5.460,148.652
C09772=1224.157,50.283,-44.598,-179.001,5.460,148.653
C09773=1224.162,50.034,-44.582,-179.003,5.459,148.654
C09774=1224.167,49.785,-44.565,-179.005,5.458,148.654
C09775=1224.172,49.535,-44.548,-179.008,5.457,148.655
C09776=1224.177,49.286,-44.533,-179.011,5.457,148.655
C09777=1224.182,49.036,-44.516,-179.013,5.456,148.656
C09778=1224.187,48.788,-44.500,-179.016,5.456,148.657
C09779=1224.192,48.538,-44.482,-179.019,5.455,148.657
C09780=1224.197,48.288,-44.466,-179.021,5.455,148.658
C09781=1224.202,48.039,-44.450,-179.023,5.454,148.658
C09782=1224.206,47.789,-44.433,-179.026,5.453,148.659
C09783=1224.212,47.540,-44.418,-179.029,5.453,148.660
C09784=1224.216,47.290,-44.401,-179.031,5.453,148.660
C09785=1224.221,47.041,-44.384,-179.033,5.452,148.661
C09786=1224.227,46.791,-44.368,-179.036,5.452,148.662
C09787=1224.231,46.542,-44.352,-179.039,5.451,148.662
C09788=1224.236,46.293,-44.335,-179.041,5.451,148.663
C09789=1224.241,46.043,-44.319,-179.043,5.450,148.664
C09790=1224.246,45.794,-44.303,-179.046,5.449,148.664
C09791=1224.251,45.545,-44.286,-179.049,5.449,148.665
C09792=1224.256,45.295,-44.271,-179.051,5.448,148.666
C09793=1224.261,45.046,-44.254,-179.054,5.447,148.666
C09794=1224.266,44.796,-44.239,-179.057,5.447,148.667
C09795=1224.270,44.547,-44.222,-179.059,5.446,148.668
C09796=1224.276,44.298,-44.206,-179.062,5.446,148.668
C09797=1224.281,44.048,-44.189,-179.064,5.445,148.669
C09798=1224.286,43.799,-44.173,-179.066,5.445,148.669
C09799=1224.291,43.549,-44.157,-179.069,5.445,148.670
C09800=1224.296,43.300,-44.140,-179.071,5.444,148.671
C09801=1224.301,43.050,-44.124,-179.074,5.443,148.671
C09802=1224.306,42.801,-44.108,-179.077,5.443,148.672
C09803=1224.311,42.551,-44.092,-179.079,5.442,148.673
C09804=1224.316,42.302,-44.076,-179.082,5.442,148.673
C09805=1224.320,42.053,-44.059,-179.084,5.441,148.674
C09806=1224.326,41.803,-44.044,-179.087,5.440,148.675
C09807=1224.330,41.554,-44.027,-179.089,5.440,148.675
C09808=1224.335,41.304,-44.011,-179.092,5.439,148.676
C09809=1224.340,41.054,-43.995,-179.095,5.439,148.677
C09810=1224.345,40.806,-43.979,-179.097,5.438,148.677
C09811=1224.350,40.555,-43.963,-179.099,5.438,148.678
C09812=1224.355,40.307,-43.947,-179.102,5.438,148.679
C09813=1224.360,40.057,-43.931,-179.105,5.437,148.679
C09814=1224.365,39.808,-43.915,-179.107,5.436,148.680
C09815=1224.370,39.558,-43.899,-179.109,5.436,148.680
C09816=1224.375,39.309,-43.882,-179.112,5.435,148.681
C09817=1224.380,39.060,-43.867,-179.115,5.435,148.682
C09818=1224.385,38.809,-43.851,-179.117,5.434,148.682
C09819=1224.389,38.561,-43.835,-179.120,5.434,148.683
C09820=1224.394,38.311,-43.819,-179.123,5.433,148.684
C09821=1224.399,38.062,-43.803,-179.125,5.433,148.684
C09822=1224.404,37.812,-43.787,-179.127,5.433,148.685
C09823=1224.409,37.563,-43.771,-179.129,5.432,148.686
C09824=1224.415,37.314,-43.755,-179.132,5.431,148.686
C09825=1224.419,37.064,-43.739,-179.135,5.431,148.687
C09826=1224.425,36.814,-43.723,-179.137,5.430,148.688
C09827=1224.429,36.565,-43.707,-179.140,5.430,148.688
C09828=1224.435,36.315,-43.691,-179.143,5.429,148.689
C09829=1224.440,36.066,-43.676,-179.145,5.428,148.690
C09830=1224.444,35.817,-43.660,-179.147,5.429,148.690
C09831=1224.449,35.567,-43.644,-179.150,5.428,148.691
C09832=1224.455,35.318,-43.628,-179.153,5.428,148.692
C09833=1224.459,35.068,-43.612,-179.155,5.427,148.692
C09834=1224.464,34.819,-43.596,-179.157,5.426,148.693
C09835=1224.469,34.569,-43.580,-179.160,5.426,148.693
C09836=1224.475,34.320,-43.565,-179.163,5.425,148.694
C09837=1224.479,34.071,-43.549,-179.165,5.425,148.695
C09838=1224.484,33.821,-43.533,-179.168,5.424,148.695
C09839=1224.489,33.572,-43.517,-179.170,5.424,148.696
C09840=1224.494,33.322,-43.502,-179.173,5.424,148.697
C09841=1224.499,33.072,-43.486,-179.175,5.423,148.698
C09842=1224.504,32.824,-43.470,-179.178,5.423,148.698
C09843=1224.509,32.574,-43.455,-179.181,5.422,148.699
C09844=1224.514,32.324,-43.439,-179.183,5.421,148.699
C09845=1224.519,32.075,-43.423,-179.185,5.421,148.700
C09846=1224.525,31.825,-43.407,-179.188,5.420,148.701
C09847=1224.528,31.576,-43.391,-179.190,5.420,148.701
C09848=1224.534,31.327,-43.376,-179.193,5.420,148.702
C09849=1224.539,31.077,-43.360,-179.195,5.419,148.703
C09850=1224.544,30.827,-43.344,-179.198,5.419,148.703
C09851=1224.548,30.578,-43.329,-179.201,5.418,148.704
C09852=1224.554,30.329,-43.314,-179.203,5.418,148.705
C09853=1224.559,30.079,-43.298,-179.206,5.417,148.705
C09854=1224.564,29.810,-43.281,-179.209,5.416,148.706
C09855=1224.569,29.542,-43.264,-179.211,5.416,148.707
C09856=1224.575,29.274,-43.247,-179.214,5.415,148.707
C09857=1224.580,29.005,-43.230,-179.217,5.415,148.708
C09858=1224.585,28.755,-43.214,-179.219,5.414,148.709
C09859=1224.590,28.506,-43.199,-179.221,5.415,148.710
C09860=1224.595,28.256,-43.184,-179.224,5.414,148.710
C09861=1224.600,28.007,-43.168,-179.227,5.413,148.711
C09862=1224.604,27.757,-43.153,-179.229,5.413,148.712
C09863=1224.610,27.508,-43.137,-179.232,5.412,148.712
C09864=1224.615,27.258,-43.122,-179.235,5.412,148.713
C09865=1224.620,27.009,-43.107,-179.237,5.411,148.714
C09866=1224.625,26.759,-43.091,-179.239,5.412,148.714
C09867=1224.630,26.510,-43.075,-179.242,5.411,148.715
C09868=1224.635,26.261,-43.060,-179.244,5.410,148.715
C09869=1224.640,26.011,-43.044,-179.247,5.410,148.716
C09870=1224.645,25.761,-43.028,-179.249,5.409,148.717
C09871=1224.649,25.512,-43.013,-179.252,5.408,148.717
C09872=1224.655,25.263,-42.998,-179.254,5.409,148.718
C09873=1224.660,25.013,-42.982,-179.257,5.408,148.719
C09874=1224.664,24.764,-42.967,-179.259,5.408,148.719
C09875=1224.670,24.514,-42.951,-179.262,5.407,148.720
C09876=1224.674,24.265,-42.936,-179.265,5.407,148.721
C09877=1224.680,24.016,-42.921,-179.267,5.406,148.722
C09878=1224.685,23.766,-42.905,-179.269,5.406,148.722
C09879=1224.689,23.516,-42.891,-179.272,5.406,148.723
C09880=1224.695,23.266,-42.875,-179.275,5.405,148.724
C09881=1224.699,23.017,-42.860,-179.277,5.405,148.724
C09882=1224.705,22.768,-42.844,-179.280,5.404,148.725
C09883=1224.710,22.518,-42.828,-179.282,5.403,148.725
C09884=1224.714,22.269,-42.813,-179.284,5.404,148.726
C09885=1224.720,22.019,-42.798,-179.287,5.403,148.727
C09886=1224.724,21.770,-42.783,-179.289,5.402,148.727
C09887=1224.730,21.520,-42.768,-179.292,5.402,148.728
C09888=1224.735,21.271,-42.753,-179.295,5.401,148.729
C09889=1224.739,21.021,-42.737,-179.297,5.401,148.729
C09890=1224.744,20.772,-42.722,-179.300,5.401,148.730
C09891=1224.750,20.523,-42.706,-179.302,5.401,148.731
C09892=1224.754,20.273,-42.691,-179.305,5.400,148.731
C09893=1224.760,20.023,-42.677,-179.307,5.399,148.732
C09894=1224.764,19.774,-42.662,-179.310,5.399,148.733
C09895=1224.769,19.524,-42.646,-179.313,5.398,148.734
C09896=1224.774,19.275,-42.631,-179.315,5.399,148.734
C09897=1224.780,19.025,-42.616,-179.317,5.398,148.735
C09898=1224.784,18.776,-42.601,-179.320,5.398,148.736
C09899=1224.790,18.527,-42.585,-179.323,5.397,148.736
C09900=1224.794,18.278,-42.570,-179.325,5.397,148.737
C09901=1224.800,18.028,-42.555,-179.327,5.396,148.737
C09902=1224.805,17.778,-42.540,-179.330,5.396,148.738
C09903=1224.809,17.528,-42.524,-179.332,5.395,148.739
C09904=1224.814,17.279,-42.509,-179.335,5.395,148.739
C09905=1224.820,17.029,-42.494,-179.338,5.394,148.740
C09906=1224.824,16.780,-42.480,-179.340,5.394,148.741
C09907=1224.829,16.531,-42.465,-179.342,5.394,148.742
C09908=1224.835,16.281,-42.450,-179.345,5.394,148.742
C09909=1224.839,16.032,-42.435,-179.348,5.393,148.743
C09910=1224.845,15.783,-42.419,-179.350,5.392,148.744
C09911=1224.850,15.533,-42.405,-179.353,5.392,148.744
C09912=1224.854,15.284,-42.390,-179.355,5.392,148.745
C09913=1224.859,15.034,-42.374,-179.358,5.392,148.746
C09914=1224.864,14.784,-42.360,-179.360,5.391,148.746
C09915=1224.870,14.535,-42.344,-179.363,5.391,148.747
C09916=1224.874,14.285,-42.330,-179.366,5.390,148.748
C09917=1224.879,14.036,-42.315,-179.368,5.390,148.748
C09918=1224.885,13.786,-42.299,-179.370,5.390,148.749
C09919=1224.889,13.537,-42.285,-179.373,5.389,148.750
C09920=1224.895,13.287,-42.269,-179.376,5.389,148.750
C09921=1224.900,13.037,-42.255,-179.378,5.388,148.751
C09922=1224.904,12.788,-42.240,-179.380,5.389,148.752
C09923=1224.910,12.538,-42.225,-179.382,5.388,148.752
C09924=1224.915,12.289,-42.210,-179.385,5.387,148.753
C09925=1224.919,12.040,-42.195,-179.388,5.387,148.754
C09926=1224.925,11.790,-42.180,-179.390,5.386,148.754
C09927=1224.930,11.541,-42.165,-179.392,5.386,148.755
C09928=1224.935,11.291,-42.151,-179.395,5.386,148.756
C09929=1224.940,11.042,-42.135,-179.398,5.385,148.756
C09930=1224.945,10.792,-42.121,-179.400,5.385,148.757
C09931=1224.950,10.543,-42.106,-179.402,5.385,148.758
C09932=1224.955,10.293,-42.092,-179.405,5.384,148.758
C09933=1224.960,10.044,-42.076,-179.408,5.384,148.759
C09934=1224.965,9.794,-42.062,-179.410,5.383,148.760
C09935=1224.970,9.545,-42.048,-179.413,5.383,148.760
C09936=1224.975,9.295,-42.032,-179.415,5.383,148.761
C09937=1224.980,9.046,-42.018,-179.418,5.383,148.762
C09938=1224.985,8.796,-42.003,-179.420,5.382,148.763
C09939=1224.990,8.547,-41.989,-179.423,5.382,148.763
C09940=1224.995,8.297,-41.973,-179.425,5.382,148.764
C09941=1225.000,8.048,-41.959,-179.428,5.381,148.765
C09942=1225.005,7.798,-41.944,-179.431,5.381,148.765
C09943=1225.010,7.549,-41.929,-179.433,5.380,148.766
C09944=1225.015,7.299,-41.915,-179.436,5.380,148.767
C09945=1225.020,7.050,-41.900,-179.438,5.380,148.767
C09946=1225.025,6.800,-41.885,-179.441,5.379,148.768
C09947=1225.030,6.550,-41.871,-179.443,5.379,148.769
C09948=1225.035,6.301,-41.856,-179.446,5.378,148.769
C09949=1225.040,6.051,-41.841,-179.448,5.379,148.770
C09950=1225.045,5.801,-41.827,-179.451,5.378,148.771
C09951=1225.050,5.552,-41.812,-179.453,5.378,148.771
C09952=1225.055,5.303,-41.798,-179.456,5.377,148.772
C09953=1225.060,5.053,-41.783,-179.457,5.377,148.773
C09954=1225.065,4.804,-41.768,-179.460,5.377,148.773
C09955=1225.070,4.554,-41.753,-179.463,5.376,148.774
C09956=1225.075,4.304,-41.739,-179.465,5.375,148.775
C09957=1225.080,4.055,-41.724,-179.468,5.375,148.775
C09958=1225.085,3.786,-41.709,-179.471,5.376,148.776
C09959=1225.091,3.518,-41.694,-179.473,5.375,148.777
C09960=1225.097,3.248,-41.678,-179.476,5.375,148.778
C09961=1225.102,2.980,-41.662,-179.479,5.374,148.778
C09962=1225.107,2.730,-41.648,-179.481,5.374,148.779
C09963=1225.112,2.480,-41.633,-179.484,5.373,148.780
C09964=1225.117,2.230,-41.619,-179.486,5.373,148.780
C09965=1225.122,1.981,-41.604,-179.489,5.373,148.781
C09966=1225.127,1.732,-41.590,-179.491,5.372,148.782
C09967=1225.132,1.482,-41.575,-179.494,5.372,148.782
C09968=1225.138,1.233,-41.561,-179.496,5.372,148.783
C09969=1225.142,0.984,-41.546,-179.499,5.372,148.784
C09970=1225.147,0.734,-41.532,-179.501,5.371,148.784
C09971=1225.152,0.484,-41.517,-179.504,5.370,148.785
C09972=1225.157,0.234,-41.503,-179.506,5.371,148.786
C09973=1225.162,-0.015,-41.489,-179.509,5.370,148.787
C09974=1225.167,-0.265,-41.475,-179.511,5.370,148.787
C09975=1225.172,-0.514,-41.460,-179.514,5.369,148.788
C09976=1225.177,-0.763,-41.446,-179.516,5.369,148.789
C09977=1225.182,-1.013,-41.431,-179.519,5.369,148.789
C09978=1225.187,-1.263,-41.417,-179.521,5.368,148.790
C09979=1225.192,-1.512,-41.403,-179.524,5.368,148.791
C09980=1225.197,-1.762,-41.389,-179.526,5.368,148.791
C09981=1225.202,-2.012,-41.374,-179.529,5.368,148.792
C09982=1225.208,-2.261,-41.360,-179.531,5.367,148.793
C09983=1225.213,-2.510,-41.346,-179.533,5.367,148.793
C09984=1225.218,-2.760,-41.332,-179.536,5.367,148.794
C09985=1225.222,-3.009,-41.317,-179.539,5.366,148.795
C09986=1225.227,-3.259,-41.303,-179.541,5.366,148.796
C09987=1225.232,-3.509,-41.288,-179.544,5.366,148.796
C09988=1225.238,-3.758,-41.274,-179.546,5.366,148.797
C09989=1225.243,-4.007,-41.260,-179.549,5.365,148.798
C09990=1225.248,-4.257,-41.246,-179.551,5.365,148.798
C09991=1225.253,-4.507,-41.232,-179.554,5.365,148.799
C09992=1225.258,-4.756,-41.217,-179.556,5.364,148.800
C09993=1225.263,-5.005,-41.203,-179.559,5.364,148.800
C09994=1225.268,-5.255,-41.189,-179.562,5.363,148.801
C09995=1225.273,-5.505,-41.175,-179.564,5.364,148.802
C09996=1225.278,-5.755,-41.161,-179.566,5.363,148.802
//INST
///DATE 2021/06/15 17:22
///ATTR SC,RW,RJ
////FRAME ROBOT
///GROUP1 RB1
NOP
MOVL C00000 V=800.0 PL=0
MOVL C00001 V=800.0 PL=0
MOVL C00002 V=800.0 PL=0
MOVL C00003 V=800.0 PL=0
MOVL C00004 V=800.0 PL=0
MOVL C00005 V=800.0 PL=0
MOVL C00006 V=800.0 PL=0
MOVL C00007 V=800.0 PL=0
MOVL C00008 V=800.0 PL=0
MOVL C00009 V=800.0 PL=0
MOVL C00010 V=800.0 PL=0
MOVL C00011 V=800.0 PL=0
MOVL C00012 V=800.0 PL=0
MOVL C00013 V=800.0 PL=0
MOVL C00014 V=800.0 PL=0
MOVL C00015 V=800.0 PL=0
MOVL C00016 V=800.0 PL=0
MOVL C00017 V=800.0 PL=0
MOVL C00018 V=800.0 PL=0
MOVL C00019 V=800.0 PL=0
MOVL C00020 V=800.0 PL=0
MOVL C00021 V=800.0 PL=0
MOVL C00022 V=800.0 PL=0
MOVL C00023 V=800.0 PL=0
MOVL C00024 V=800.0 PL=0
MOVL C00025 V=800.0 PL=0
MOVL C00026 V=800.0 PL=0
MOVL C00027 V=800.0 PL=0
MOVL C00028 V=800.0 PL=0
MOVL C00029 V=800.0 PL=0
MOVL C00030 V=800.0 PL=0
MOVL C00031 V=800.0 PL=0
MOVL C00032 V=800.0 PL=0
MOVL C00033 V=800.0 PL=0
MOVL C00034 V=800.0 PL=0
MOVL C00035 V=800.0 PL=0
MOVL C00036 V=800.0 PL=0
MOVL C00037 V=800.0 PL=0
MOVL C00038 V=800.0 PL=0
MOVL C00039 V=800.0 PL=0
MOVL C00040 V=800.0 PL=0
MOVL C00041 V=800.0 PL=0
MOVL C00042 V=800.0 PL=0
MOVL C00043 V=800.0 PL=0
MOVL C00044 V=800.0 PL=0
MOVL C00045 V=800.0 PL=0
MOVL C00046 V=800.0 PL=0
MOVL C00047 V=800.0 PL=0
MOVL C00048 V=800.0 PL=0
MOVL C00049 V=800.0 PL=0
MOVL C00050 V=800.0 PL=0
MOVL C00051 V=800.0 PL=0
MOVL C00052 V=800.0 PL=0
MOVL C00053 V=800.0 PL=0
MOVL C00054 V=800.0 PL=0
MOVL C00055 V=800.0 PL=0
MOVL C00056 V=800.0 PL=0
MOVL C00057 V=800.0 PL=0
MOVL C00058 V=800.0 PL=0
MOVL C00059 V=800.0 PL=0
MOVL C00060 V=800.0 PL=0
MOVL C00061 V=800.0 PL=0
MOVL C00062 V=800.0 PL=0
MOVL C00063 V=800.0 PL=0
MOVL C00064 V=800.0 PL=0
MOVL C00065 V=800.0 PL=0
MOVL C00066 V=800.0 PL=0
MOVL C00067 V=800.0 PL=0
MOVL C00068 V=800.0 PL=0
MOVL C00069 V=800.0 PL=0
MOVL C00070 V=800.0 PL=0
MOVL C00071 V=800.0 PL=0
MOVL C00072 V=800.0 PL=0
MOVL C00073 V=800.0 PL=0
MOVL C00074 V=800.0 PL=0
MOVL C00075 V=800.0 PL=0
MOVL C00076 V=800.0 PL=0
MOVL C00077 V=800.0 PL=0
MOVL C00078 V=800.0 PL=0
MOVL C00079 V=800.0 PL=0
MOVL C00080 V=800.0 PL=0
MOVL C00081 V=800.0 PL=0
MOVL C00082 V=800.0 PL=0
MOVL C00083 V=800.0 PL=0
MOVL C00084 V=800.0 PL=0
MOVL C00085 V=800.0 PL=0
MOVL C00086 V=800.0 PL=0
MOVL C00087 V=800.0 PL=0
MOVL C00088 V=800.0 PL=0
MOVL C00089 V=800.0 PL=0
MOVL C00090 V=800.0 PL=0
MOVL C00091 V=800.0 PL=0
MOVL C00092 V=800.0 PL=0
MOVL C00093 V=800.0 PL=0
MOVL C00094 V=800.0 PL=0
MOVL C00095 V=800.0 PL=0
MOVL C00096 V=800.0 PL=0
MOVL C00097 V=800.0 PL=0
MOVL C00098 V=800.0 PL=0
MOVL C00099 V=800.0 PL=0
MOVL C00100 V=800.0 PL=0
MOVL C00101 V=800.0 PL=0
MOVL C00102 V=800.0 PL=0
MOVL C00103 V=800.0 PL=0
MOVL C00104 V=800.0 PL=0
MOVL C00105 V=800.0 PL=0
MOVL C00106 V=800.0 PL=0
MOVL C00107 V=800.0 PL=0
MOVL C00108 V=800.0 PL=0
MOVL C00109 V=800.0 PL=0
MOVL C00110 V=800.0 PL=0
MOVL C00111 V=800.0 PL=0
MOVL C00112 V=800.0 PL=0
MOVL C00113 V=800.0 PL=0
MOVL C00114 V=800.0 PL=0
MOVL C00115 V=800.0 PL=0
MOVL C00116 V=800.0 PL=0
MOVL C00117 V=800.0 PL=0
MOVL C00118 V=800.0 PL=0
MOVL C00119 V=800.0 PL=0
MOVL C00120 V=800.0 PL=0
MOVL C00121 V=800.0 PL=0
MOVL C00122 V=800.0 PL=0
MOVL C00123 V=800.0 PL=0
MOVL C00124 V=800.0 PL=0
MOVL C00125 V=800.0 PL=0
MOVL C00126 V=800.0 PL=0
MOVL C00127 V=800.0 PL=0
MOVL C00128 V=800.0 PL=0
MOVL C00129 V=800.0 PL=0
MOVL C00130 V=800.0 PL=0
MOVL C00131 V=800.0 PL=0
MOVL C00132 V=800.0 PL=0
MOVL C00133 V=800.0 PL=0
MOVL C00134 V=800.0 PL=0
MOVL C00135 V=800.0 PL=0
MOVL C00136 V=800.0 PL=0
MOVL C00137 V=800.0 PL=0
MOVL C00138 V=800.0 PL=0
MOVL C00139 V=800.0 PL=0
MOVL C00140 V=800.0 PL=0
MOVL C00141 V=800.0 PL=0
MOVL C00142 V=800.0 PL=0
MOVL C00143 V=800.0 PL=0
MOVL C00144 V=800.0 PL=0
MOVL C00145 V=800.0 PL=0
MOVL C00146 V=800.0 PL=0
MOVL C00147 V=800.0 PL=0
MOVL C00148 V=800.0 PL=0
MOVL C00149 V=800.0 PL=0
MOVL C00150 V=800.0 PL=0
MOVL C00151 V=800.0 PL=0
MOVL C00152 V=800.0 PL=0
MOVL C00153 V=800.0 PL=0
MOVL C00154 V=800.0 PL=0
MOVL C00155 V=800.0 PL=0
MOVL C00156 V=800.0 PL=0
MOVL C00157 V=800.0 PL=0
MOVL C00158 V=800.0 PL=0
MOVL C00159 V=800.0 PL=0
MOVL C00160 V=800.0 PL=0
MOVL C00161 V=800.0 PL=0
MOVL C00162 V=800.0 PL=0
MOVL C00163 V=800.0 PL=0
MOVL C00164 V=800.0 PL=0
MOVL C00165 V=800.0 PL=0
MOVL C00166 V=800.0 PL=0
MOVL C00167 V=800.0 PL=0
MOVL C00168 V=800.0 PL=0
MOVL C00169 V=800.0 PL=0
MOVL C00170 V=800.0 PL=0
MOVL C00171 V=800.0 PL=0
MOVL C00172 V=800.0 PL=0
MOVL C00173 V=800.0 PL=0
MOVL C00174 V=800.0 PL=0
MOVL C00175 V=800.0 PL=0
MOVL C00176 V=800.0 PL=0
MOVL C00177 V=800.0 PL=0
MOVL C00178 V=800.0 PL=0
MOVL C00179 V=800.0 PL=0
MOVL C00180 V=800.0 PL=0
MOVL C00181 V=800.0 PL=0
MOVL C00182 V=800.0 PL=0
MOVL C00183 V=800.0 PL=0
MOVL C00184 V=800.0 PL=0
MOVL C00185 V=800.0 PL=0
MOVL C00186 V=800.0 PL=0
MOVL C00187 V=800.0 PL=0
MOVL C00188 V=800.0 PL=0
MOVL C00189 V=800.0 PL=0
MOVL C00190 V=800.0 PL=0
MOVL C00191 V=800.0 PL=0
MOVL C00192 V=800.0 PL=0
MOVL C00193 V=800.0 PL=0
MOVL C00194 V=800.0 PL=0
MOVL C00195 V=800.0 PL=0
MOVL C00196 V=800.0 PL=0
MOVL C00197 V=800.0 PL=0
MOVL C00198 V=800.0 PL=0
MOVL C00199 V=800.0 PL=0
MOVL C00200 V=800.0 PL=0
MOVL C00201 V=800.0 PL=0
MOVL C00202 V=800.0 PL=0
MOVL C00203 V=800.0 PL=0
MOVL C00204 V=800.0 PL=0
MOVL C00205 V=800.0 PL=0
MOVL C00206 V=800.0 PL=0
MOVL C00207 V=800.0 PL=0
MOVL C00208 V=800.0 PL=0
MOVL C00209 V=800.0 PL=0
MOVL C00210 V=800.0 PL=0
MOVL C00211 V=800.0 PL=0
MOVL C00212 V=800.0 PL=0
MOVL C00213 V=800.0 PL=0
MOVL C00214 V=800.0 PL=0
MOVL C00215 V=800.0 PL=0
MOVL C00216 V=800.0 PL=0
MOVL C00217 V=800.0 PL=0
MOVL C00218 V=800.0 PL=0
MOVL C00219 V=800.0 PL=0
MOVL C00220 V=800.0 PL=0
MOVL C00221 V=800.0 PL=0
MOVL C00222 V=800.0 PL=0
MOVL C00223 V=800.0 PL=0
MOVL C00224 V=800.0 PL=0
MOVL C00225 V=800.0 PL=0
MOVL C00226 V=800.0 PL=0
MOVL C00227 V=800.0 PL=0
MOVL C00228 V=800.0 PL=0
MOVL C00229 V=800.0 PL=0
MOVL C00230 V=800.0 PL=0
MOVL C00231 V=800.0 PL=0
MOVL C00232 V=800.0 PL=0
MOVL C00233 V=800.0 PL=0
MOVL C00234 V=800.0 PL=0
MOVL C00235 V=800.0 PL=0
MOVL C00236 V=800.0 PL=0
MOVL C00237 V=800.0 PL=0
MOVL C00238 V=800.0 PL=0
MOVL C00239 V=800.0 PL=0
MOVL C00240 V=800.0 PL=0
MOVL C00241 V=800.0 PL=0
MOVL C00242 V=800.0 PL=0
MOVL C00243 V=800.0 PL=0
MOVL C00244 V=800.0 PL=0
MOVL C00245 V=800.0 PL=0
MOVL C00246 V=800.0 PL=0
MOVL C00247 V=800.0 PL=0
MOVL C00248 V=800.0 PL=0
MOVL C00249 V=800.0 PL=0
MOVL C00250 V=800.0 PL=0
MOVL C00251 V=800.0 PL=0
MOVL C00252 V=800.0 PL=0
MOVL C00253 V=800.0 PL=0
MOVL C00254 V=800.0 PL=0
MOVL C00255 V=800.0 PL=0
MOVL C00256 V=800.0 PL=0
MOVL C00257 V=800.0 PL=0
MOVL C00258 V=800.0 PL=0
MOVL C00259 V=800.0 PL=0
MOVL C00260 V=800.0 PL=0
MOVL C00261 V=800.0 PL=0
MOVL C00262 V=800.0 PL=0
MOVL C00263 V=800.0 PL=0
MOVL C00264 V=800.0 PL=0
MOVL C00265 V=800.0 PL=0
MOVL C00266 V=800.0 PL=0
MOVL C00267 V=800.0 PL=0
MOVL C00268 V=800.0 PL=0
MOVL C00269 V=800.0 PL=0
MOVL C00270 V=800.0 PL=0
MOVL C00271 V=800.0 PL=0
MOVL C00272 V=800.0 PL=0
MOVL C00273 V=800.0 PL=0
MOVL C00274 V=800.0 PL=0
MOVL C00275 V=800.0 PL=0
MOVL C00276 V=800.0 PL=0
MOVL C00277 V=800.0 PL=0
MOVL C00278 V=800.0 PL=0
MOVL C00279 V=800.0 PL=0
MOVL C00280 V=800.0 PL=0
MOVL C00281 V=800.0 PL=0
MOVL C00282 V=800.0 PL=0
MOVL C00283 V=800.0 PL=0
MOVL C00284 V=800.0 PL=0
MOVL C00285 V=800.0 PL=0
MOVL C00286 V=800.0 PL=0
MOVL C00287 V=800.0 PL=0
MOVL C00288 V=800.0 PL=0
MOVL C00289 V=800.0 PL=0
MOVL C00290 V=800.0 PL=0
MOVL C00291 V=800.0 PL=0
MOVL C00292 V=800.0 PL=0
MOVL C00293 V=800.0 PL=0
MOVL C00294 V=800.0 PL=0
MOVL C00295 V=800.0 PL=0
MOVL C00296 V=800.0 PL=0
MOVL C00297 V=800.0 PL=0
MOVL C00298 V=800.0 PL=0
MOVL C00299 V=800.0 PL=0
MOVL C00300 V=800.0 PL=0
MOVL C00301 V=800.0 PL=0
MOVL C00302 V=800.0 PL=0
MOVL C00303 V=800.0 PL=0
MOVL C00304 V=800.0 PL=0
MOVL C00305 V=800.0 PL=0
MOVL C00306 V=800.0 PL=0
MOVL C00307 V=800.0 PL=0
MOVL C00308 V=800.0 PL=0
MOVL C00309 V=800.0 PL=0
MOVL C00310 V=800.0 PL=0
MOVL C00311 V=800.0 PL=0
MOVL C00312 V=800.0 PL=0
MOVL C00313 V=800.0 PL=0
MOVL C00314 V=800.0 PL=0
MOVL C00315 V=800.0 PL=0
MOVL C00316 V=800.0 PL=0
MOVL C00317 V=800.0 PL=0
MOVL C00318 V=800.0 PL=0
MOVL C00319 V=800.0 PL=0
MOVL C00320 V=800.0 PL=0
MOVL C00321 V=800.0 PL=0
MOVL C00322 V=800.0 PL=0
MOVL C00323 V=800.0 PL=0
MOVL C00324 V=800.0 PL=0
MOVL C00325 V=800.0 PL=0
MOVL C00326 V=800.0 PL=0
MOVL C00327 V=800.0 PL=0
MOVL C00328 V=800.0 PL=0
MOVL C00329 V=800.0 PL=0
MOVL C00330 V=800.0 PL=0
MOVL C00331 V=800.0 PL=0
MOVL C00332 V=800.0 PL=0
MOVL C00333 V=800.0 PL=0
MOVL C00334 V=800.0 PL=0
MOVL C00335 V=800.0 PL=0
MOVL C00336 V=800.0 PL=0
MOVL C00337 V=800.0 PL=0
MOVL C00338 V=800.0 PL=0
MOVL C00339 V=800.0 PL=0
MOVL C00340 V=800.0 PL=0
MOVL C00341 V=800.0 PL=0
MOVL C00342 V=800.0 PL=0
MOVL C00343 V=800.0 PL=0
MOVL C00344 V=800.0 PL=0
MOVL C00345 V=800.0 PL=0
MOVL C00346 V=800.0 PL=0
MOVL C00347 V=800.0 PL=0
MOVL C00348 V=800.0 PL=0
MOVL C00349 V=800.0 PL=0
MOVL C00350 V=800.0 PL=0
MOVL C00351 V=800.0 PL=0
MOVL C00352 V=800.0 PL=0
MOVL C00353 V=800.0 PL=0
MOVL C00354 V=800.0 PL=0
MOVL C00355 V=800.0 PL=0
MOVL C00356 V=800.0 PL=0
MOVL C00357 V=800.0 PL=0
MOVL C00358 V=800.0 PL=0
MOVL C00359 V=800.0 PL=0
MOVL C00360 V=800.0 PL=0
MOVL C00361 V=800.0 PL=0
MOVL C00362 V=800.0 PL=0
MOVL C00363 V=800.0 PL=0
MOVL C00364 V=800.0 PL=0
MOVL C00365 V=800.0 PL=0
MOVL C00366 V=800.0 PL=0
MOVL C00367 V=800.0 PL=0
MOVL C00368 V=800.0 PL=0
MOVL C00369 V=800.0 PL=0
MOVL C00370 V=800.0 PL=0
MOVL C00371 V=800.0 PL=0
MOVL C00372 V=800.0 PL=0
MOVL C00373 V=800.0 PL=0
MOVL C00374 V=800.0 PL=0
MOVL C00375 V=800.0 PL=0
MOVL C00376 V=800.0 PL=0
MOVL C00377 V=800.0 PL=0
MOVL C00378 V=800.0 PL=0
MOVL C00379 V=800.0 PL=0
MOVL C00380 V=800.0 PL=0
MOVL C00381 V=800.0 PL=0
MOVL C00382 V=800.0 PL=0
MOVL C00383 V=800.0 PL=0
MOVL C00384 V=800.0 PL=0
MOVL C00385 V=800.0 PL=0
MOVL C00386 V=800.0 PL=0
MOVL C00387 V=800.0 PL=0
MOVL C00388 V=800.0 PL=0
MOVL C00389 V=800.0 PL=0
MOVL C00390 V=800.0 PL=0
MOVL C00391 V=800.0 PL=0
MOVL C00392 V=800.0 PL=0
MOVL C00393 V=800.0 PL=0
MOVL C00394 V=800.0 PL=0
MOVL C00395 V=800.0 PL=0
MOVL C00396 V=800.0 PL=0
MOVL C00397 V=800.0 PL=0
MOVL C00398 V=800.0 PL=0
MOVL C00399 V=800.0 PL=0
MOVL C00400 V=800.0 PL=0
MOVL C00401 V=800.0 PL=0
MOVL C00402 V=800.0 PL=0
MOVL C00403 V=800.0 PL=0
MOVL C00404 V=800.0 PL=0
MOVL C00405 V=800.0 PL=0
MOVL C00406 V=800.0 PL=0
MOVL C00407 V=800.0 PL=0
MOVL C00408 V=800.0 PL=0
MOVL C00409 V=800.0 PL=0
MOVL C00410 V=800.0 PL=0
MOVL C00411 V=800.0 PL=0
MOVL C00412 V=800.0 PL=0
MOVL C00413 V=800.0 PL=0
MOVL C00414 V=800.0 PL=0
MOVL C00415 V=800.0 PL=0
MOVL C00416 V=800.0 PL=0
MOVL C00417 V=800.0 PL=0
MOVL C00418 V=800.0 PL=0
MOVL C00419 V=800.0 PL=0
MOVL C00420 V=800.0 PL=0
MOVL C00421 V=800.0 PL=0
MOVL C00422 V=800.0 PL=0
MOVL C00423 V=800.0 PL=0
MOVL C00424 V=800.0 PL=0
MOVL C00425 V=800.0 PL=0
MOVL C00426 V=800.0 PL=0
MOVL C00427 V=800.0 PL=0
MOVL C00428 V=800.0 PL=0
MOVL C00429 V=800.0 PL=0
MOVL C00430 V=800.0 PL=0
MOVL C00431 V=800.0 PL=0
MOVL C00432 V=800.0 PL=0
MOVL C00433 V=800.0 PL=0
MOVL C00434 V=800.0 PL=0
MOVL C00435 V=800.0 PL=0
MOVL C00436 V=800.0 PL=0
MOVL C00437 V=800.0 PL=0
MOVL C00438 V=800.0 PL=0
MOVL C00439 V=800.0 PL=0
MOVL C00440 V=800.0 PL=0
MOVL C00441 V=800.0 PL=0
MOVL C00442 V=800.0 PL=0
MOVL C00443 V=800.0 PL=0
MOVL C00444 V=800.0 PL=0
MOVL C00445 V=800.0 PL=0
MOVL C00446 V=800.0 PL=0
MOVL C00447 V=800.0 PL=0
MOVL C00448 V=800.0 PL=0
MOVL C00449 V=800.0 PL=0
MOVL C00450 V=800.0 PL=0
MOVL C00451 V=800.0 PL=0
MOVL C00452 V=800.0 PL=0
MOVL C00453 V=800.0 PL=0
MOVL C00454 V=800.0 PL=0
MOVL C00455 V=800.0 PL=0
MOVL C00456 V=800.0 PL=0
MOVL C00457 V=800.0 PL=0
MOVL C00458 V=800.0 PL=0
MOVL C00459 V=800.0 PL=0
MOVL C00460 V=800.0 PL=0
MOVL C00461 V=800.0 PL=0
MOVL C00462 V=800.0 PL=0
MOVL C00463 V=800.0 PL=0
MOVL C00464 V=800.0 PL=0
MOVL C00465 V=800.0 PL=0
MOVL C00466 V=800.0 PL=0
MOVL C00467 V=800.0 PL=0
MOVL C00468 V=800.0 PL=0
MOVL C00469 V=800.0 PL=0
MOVL C00470 V=800.0 PL=0
MOVL C00471 V=800.0 PL=0
MOVL C00472 V=800.0 PL=0
MOVL C00473 V=800.0 PL=0
MOVL C00474 V=800.0 PL=0
MOVL C00475 V=800.0 PL=0
MOVL C00476 V=800.0 PL=0
MOVL C00477 V=800.0 PL=0
MOVL C00478 V=800.0 PL=0
MOVL C00479 V=800.0 PL=0
MOVL C00480 V=800.0 PL=0
MOVL C00481 V=800.0 PL=0
MOVL C00482 V=800.0 PL=0
MOVL C00483 V=800.0 PL=0
MOVL C00484 V=800.0 PL=0
MOVL C00485 V=800.0 PL=0
MOVL C00486 V=800.0 PL=0
MOVL C00487 V=800.0 PL=0
MOVL C00488 V=800.0 PL=0
MOVL C00489 V=800.0 PL=0
MOVL C00490 V=800.0 PL=0
MOVL C00491 V=800.0 PL=0
MOVL C00492 V=800.0 PL=0
MOVL C00493 V=800.0 PL=0
MOVL C00494 V=800.0 PL=0
MOVL C00495 V=800.0 PL=0
MOVL C00496 V=800.0 PL=0
MOVL C00497 V=800.0 PL=0
MOVL C00498 V=800.0 PL=0
MOVL C00499 V=800.0 PL=0
MOVL C00500 V=800.0 PL=0
MOVL C00501 V=800.0 PL=0
MOVL C00502 V=800.0 PL=0
MOVL C00503 V=800.0 PL=0
MOVL C00504 V=800.0 PL=0
MOVL C00505 V=800.0 PL=0
MOVL C00506 V=800.0 PL=0
MOVL C00507 V=800.0 PL=0
MOVL C00508 V=800.0 PL=0
MOVL C00509 V=800.0 PL=0
MOVL C00510 V=800.0 PL=0
MOVL C00511 V=800.0 PL=0
MOVL C00512 V=800.0 PL=0
MOVL C00513 V=800.0 PL=0
MOVL C00514 V=800.0 PL=0
MOVL C00515 V=800.0 PL=0
MOVL C00516 V=800.0 PL=0
MOVL C00517 V=800.0 PL=0
MOVL C00518 V=800.0 PL=0
MOVL C00519 V=800.0 PL=0
MOVL C00520 V=800.0 PL=0
MOVL C00521 V=800.0 PL=0
MOVL C00522 V=800.0 PL=0
MOVL C00523 V=800.0 PL=0
MOVL C00524 V=800.0 PL=0
MOVL C00525 V=800.0 PL=0
MOVL C00526 V=800.0 PL=0
MOVL C00527 V=800.0 PL=0
MOVL C00528 V=800.0 PL=0
MOVL C00529 V=800.0 PL=0
MOVL C00530 V=800.0 PL=0
MOVL C00531 V=800.0 PL=0
MOVL C00532 V=800.0 PL=0
MOVL C00533 V=800.0 PL=0
MOVL C00534 V=800.0 PL=0
MOVL C00535 V=800.0 PL=0
MOVL C00536 V=800.0 PL=0
MOVL C00537 V=800.0 PL=0
MOVL C00538 V=800.0 PL=0
MOVL C00539 V=800.0 PL=0
MOVL C00540 V=800.0 PL=0
MOVL C00541 V=800.0 PL=0
MOVL C00542 V=800.0 PL=0
MOVL C00543 V=800.0 PL=0
MOVL C00544 V=800.0 PL=0
MOVL C00545 V=800.0 PL=0
MOVL C00546 V=800.0 PL=0
MOVL C00547 V=800.0 PL=0
MOVL C00548 V=800.0 PL=0
MOVL C00549 V=800.0 PL=0
MOVL C00550 V=800.0 PL=0
MOVL C00551 V=800.0 PL=0
MOVL C00552 V=800.0 PL=0
MOVL C00553 V=800.0 PL=0
MOVL C00554 V=800.0 PL=0
MOVL C00555 V=800.0 PL=0
MOVL C00556 V=800.0 PL=0
MOVL C00557 V=800.0 PL=0
MOVL C00558 V=800.0 PL=0
MOVL C00559 V=800.0 PL=0
MOVL C00560 V=800.0 PL=0
MOVL C00561 V=800.0 PL=0
MOVL C00562 V=800.0 PL=0
MOVL C00563 V=800.0 PL=0
MOVL C00564 V=800.0 PL=0
MOVL C00565 V=800.0 PL=0
MOVL C00566 V=800.0 PL=0
MOVL C00567 V=800.0 PL=0
MOVL C00568 V=800.0 PL=0
MOVL C00569 V=800.0 PL=0
MOVL C00570 V=800.0 PL=0
MOVL C00571 V=800.0 PL=0
MOVL C00572 V=800.0 PL=0
MOVL C00573 V=800.0 PL=0
MOVL C00574 V=800.0 PL=0
MOVL C00575 V=800.0 PL=0
MOVL C00576 V=800.0 PL=0
MOVL C00577 V=800.0 PL=0
MOVL C00578 V=800.0 PL=0
MOVL C00579 V=800.0 PL=0
MOVL C00580 V=800.0 PL=0
MOVL C00581 V=800.0 PL=0
MOVL C00582 V=800.0 PL=0
MOVL C00583 V=800.0 PL=0
MOVL C00584 V=800.0 PL=0
MOVL C00585 V=800.0 PL=0
MOVL C00586 V=800.0 PL=0
MOVL C00587 V=800.0 PL=0
MOVL C00588 V=800.0 PL=0
MOVL C00589 V=800.0 PL=0
MOVL C00590 V=800.0 PL=0
MOVL C00591 V=800.0 PL=0
MOVL C00592 V=800.0 PL=0
MOVL C00593 V=800.0 PL=0
MOVL C00594 V=800.0 PL=0
MOVL C00595 V=800.0 PL=0
MOVL C00596 V=800.0 PL=0
MOVL C00597 V=800.0 PL=0
MOVL C00598 V=800.0 PL=0
MOVL C00599 V=800.0 PL=0
MOVL C00600 V=800.0 PL=0
MOVL C00601 V=800.0 PL=0
MOVL C00602 V=800.0 PL=0
MOVL C00603 V=800.0 PL=0
MOVL C00604 V=800.0 PL=0
MOVL C00605 V=800.0 PL=0
MOVL C00606 V=800.0 PL=0
MOVL C00607 V=800.0 PL=0
MOVL C00608 V=800.0 PL=0
MOVL C00609 V=800.0 PL=0
MOVL C00610 V=800.0 PL=0
MOVL C00611 V=800.0 PL=0
MOVL C00612 V=800.0 PL=0
MOVL C00613 V=800.0 PL=0
MOVL C00614 V=800.0 PL=0
MOVL C00615 V=800.0 PL=0
MOVL C00616 V=800.0 PL=0
MOVL C00617 V=800.0 PL=0
MOVL C00618 V=800.0 PL=0
MOVL C00619 V=800.0 PL=0
MOVL C00620 V=800.0 PL=0
MOVL C00621 V=800.0 PL=0
MOVL C00622 V=800.0 PL=0
MOVL C00623 V=800.0 PL=0
MOVL C00624 V=800.0 PL=0
MOVL C00625 V=800.0 PL=0
MOVL C00626 V=800.0 PL=0
MOVL C00627 V=800.0 PL=0
MOVL C00628 V=800.0 PL=0
MOVL C00629 V=800.0 PL=0
MOVL C00630 V=800.0 PL=0
MOVL C00631 V=800.0 PL=0
MOVL C00632 V=800.0 PL=0
MOVL C00633 V=800.0 PL=0
MOVL C00634 V=800.0 PL=0
MOVL C00635 V=800.0 PL=0
MOVL C00636 V=800.0 PL=0
MOVL C00637 V=800.0 PL=0
MOVL C00638 V=800.0 PL=0
MOVL C00639 V=800.0 PL=0
MOVL C00640 V=800.0 PL=0
MOVL C00641 V=800.0 PL=0
MOVL C00642 V=800.0 PL=0
MOVL C00643 V=800.0 PL=0
MOVL C00644 V=800.0 PL=0
MOVL C00645 V=800.0 PL=0
MOVL C00646 V=800.0 PL=0
MOVL C00647 V=800.0 PL=0
MOVL C00648 V=800.0 PL=0
MOVL C00649 V=800.0 PL=0
MOVL C00650 V=800.0 PL=0
MOVL C00651 V=800.0 PL=0
MOVL C00652 V=800.0 PL=0
MOVL C00653 V=800.0 PL=0
MOVL C00654 V=800.0 PL=0
MOVL C00655 V=800.0 PL=0
MOVL C00656 V=800.0 PL=0
MOVL C00657 V=800.0 PL=0
MOVL C00658 V=800.0 PL=0
MOVL C00659 V=800.0 PL=0
MOVL C00660 V=800.0 PL=0
MOVL C00661 V=800.0 PL=0
MOVL C00662 V=800.0 PL=0
MOVL C00663 V=800.0 PL=0
MOVL C00664 V=800.0 PL=0
MOVL C00665 V=800.0 PL=0
MOVL C00666 V=800.0 PL=0
MOVL C00667 V=800.0 PL=0
MOVL C00668 V=800.0 PL=0
MOVL C00669 V=800.0 PL=0
MOVL C00670 V=800.0 PL=0
MOVL C00671 V=800.0 PL=0
MOVL C00672 V=800.0 PL=0
MOVL C00673 V=800.0 PL=0
MOVL C00674 V=800.0 PL=0
MOVL C00675 V=800.0 PL=0
MOVL C00676 V=800.0 PL=0
MOVL C00677 V=800.0 PL=0
MOVL C00678 V=800.0 PL=0
MOVL C00679 V=800.0 PL=0
MOVL C00680 V=800.0 PL=0
MOVL C00681 V=800.0 PL=0
MOVL C00682 V=800.0 PL=0
MOVL C00683 V=800.0 PL=0
MOVL C00684 V=800.0 PL=0
MOVL C00685 V=800.0 PL=0
MOVL C00686 V=800.0 PL=0
MOVL C00687 V=800.0 PL=0
MOVL C00688 V=800.0 PL=0
MOVL C00689 V=800.0 PL=0
MOVL C00690 V=800.0 PL=0
MOVL C00691 V=800.0 PL=0
MOVL C00692 V=800.0 PL=0
MOVL C00693 V=800.0 PL=0
MOVL C00694 V=800.0 PL=0
MOVL C00695 V=800.0 PL=0
MOVL C00696 V=800.0 PL=0
MOVL C00697 V=800.0 PL=0
MOVL C00698 V=800.0 PL=0
MOVL C00699 V=800.0 PL=0
MOVL C00700 V=800.0 PL=0
MOVL C00701 V=800.0 PL=0
MOVL C00702 V=800.0 PL=0
MOVL C00703 V=800.0 PL=0
MOVL C00704 V=800.0 PL=0
MOVL C00705 V=800.0 PL=0
MOVL C00706 V=800.0 PL=0
MOVL C00707 V=800.0 PL=0
MOVL C00708 V=800.0 PL=0
MOVL C00709 V=800.0 PL=0
MOVL C00710 V=800.0 PL=0
MOVL C00711 V=800.0 PL=0
MOVL C00712 V=800.0 PL=0
MOVL C00713 V=800.0 PL=0
MOVL C00714 V=800.0 PL=0
MOVL C00715 V=800.0 PL=0
MOVL C00716 V=800.0 PL=0
MOVL C00717 V=800.0 PL=0
MOVL C00718 V=800.0 PL=0
MOVL C00719 V=800.0 PL=0
MOVL C00720 V=800.0 PL=0
MOVL C00721 V=800.0 PL=0
MOVL C00722 V=800.0 PL=0
MOVL C00723 V=800.0 PL=0
MOVL C00724 V=800.0 PL=0
MOVL C00725 V=800.0 PL=0
MOVL C00726 V=800.0 PL=0
MOVL C00727 V=800.0 PL=0
MOVL C00728 V=800.0 PL=0
MOVL C00729 V=800.0 PL=0
MOVL C00730 V=800.0 PL=0
MOVL C00731 V=800.0 PL=0
MOVL C00732 V=800.0 PL=0
MOVL C00733 V=800.0 PL=0
MOVL C00734 V=800.0 PL=0
MOVL C00735 V=800.0 PL=0
MOVL C00736 V=800.0 PL=0
MOVL C00737 V=800.0 PL=0
MOVL C00738 V=800.0 PL=0
MOVL C00739 V=800.0 PL=0
MOVL C00740 V=800.0 PL=0
MOVL C00741 V=800.0 PL=0
MOVL C00742 V=800.0 PL=0
MOVL C00743 V=800.0 PL=0
MOVL C00744 V=800.0 PL=0
MOVL C00745 V=800.0 PL=0
MOVL C00746 V=800.0 PL=0
MOVL C00747 V=800.0 PL=0
MOVL C00748 V=800.0 PL=0
MOVL C00749 V=800.0 PL=0
MOVL C00750 V=800.0 PL=0
MOVL C00751 V=800.0 PL=0
MOVL C00752 V=800.0 PL=0
MOVL C00753 V=800.0 PL=0
MOVL C00754 V=800.0 PL=0
MOVL C00755 V=800.0 PL=0
MOVL C00756 V=800.0 PL=0
MOVL C00757 V=800.0 PL=0
MOVL C00758 V=800.0 PL=0
MOVL C00759 V=800.0 PL=0
MOVL C00760 V=800.0 PL=0
MOVL C00761 V=800.0 PL=0
MOVL C00762 V=800.0 PL=0
MOVL C00763 V=800.0 PL=0
MOVL C00764 V=800.0 PL=0
MOVL C00765 V=800.0 PL=0
MOVL C00766 V=800.0 PL=0
MOVL C00767 V=800.0 PL=0
MOVL C00768 V=800.0 PL=0
MOVL C00769 V=800.0 PL=0
MOVL C00770 V=800.0 PL=0
MOVL C00771 V=800.0 PL=0
MOVL C00772 V=800.0 PL=0
MOVL C00773 V=800.0 PL=0
MOVL C00774 V=800.0 PL=0
MOVL C00775 V=800.0 PL=0
MOVL C00776 V=800.0 PL=0
MOVL C00777 V=800.0 PL=0
MOVL C00778 V=800.0 PL=0
MOVL C00779 V=800.0 PL=0
MOVL C00780 V=800.0 PL=0
MOVL C00781 V=800.0 PL=0
MOVL C00782 V=800.0 PL=0
MOVL C00783 V=800.0 PL=0
MOVL C00784 V=800.0 PL=0
MOVL C00785 V=800.0 PL=0
MOVL C00786 V=800.0 PL=0
MOVL C00787 V=800.0 PL=0
MOVL C00788 V=800.0 PL=0
MOVL C00789 V=800.0 PL=0
MOVL C00790 V=800.0 PL=0
MOVL C00791 V=800.0 PL=0
MOVL C00792 V=800.0 PL=0
MOVL C00793 V=800.0 PL=0
MOVL C00794 V=800.0 PL=0
MOVL C00795 V=800.0 PL=0
MOVL C00796 V=800.0 PL=0
MOVL C00797 V=800.0 PL=0
MOVL C00798 V=800.0 PL=0
MOVL C00799 V=800.0 PL=0
MOVL C00800 V=800.0 PL=0
MOVL C00801 V=800.0 PL=0
MOVL C00802 V=800.0 PL=0
MOVL C00803 V=800.0 PL=0
MOVL C00804 V=800.0 PL=0
MOVL C00805 V=800.0 PL=0
MOVL C00806 V=800.0 PL=0
MOVL C00807 V=800.0 PL=0
MOVL C00808 V=800.0 PL=0
MOVL C00809 V=800.0 PL=0
MOVL C00810 V=800.0 PL=0
MOVL C00811 V=800.0 PL=0
MOVL C00812 V=800.0 PL=0
MOVL C00813 V=800.0 PL=0
MOVL C00814 V=800.0 PL=0
MOVL C00815 V=800.0 PL=0
MOVL C00816 V=800.0 PL=0
MOVL C00817 V=800.0 PL=0
MOVL C00818 V=800.0 PL=0
MOVL C00819 V=800.0 PL=0
MOVL C00820 V=800.0 PL=0
MOVL C00821 V=800.0 PL=0
MOVL C00822 V=800.0 PL=0
MOVL C00823 V=800.0 PL=0
MOVL C00824 V=800.0 PL=0
MOVL C00825 V=800.0 PL=0
MOVL C00826 V=800.0 PL=0
MOVL C00827 V=800.0 PL=0
MOVL C00828 V=800.0 PL=0
MOVL C00829 V=800.0 PL=0
MOVL C00830 V=800.0 PL=0
MOVL C00831 V=800.0 PL=0
MOVL C00832 V=800.0 PL=0
MOVL C00833 V=800.0 PL=0
MOVL C00834 V=800.0 PL=0
MOVL C00835 V=800.0 PL=0
MOVL C00836 V=800.0 PL=0
MOVL C00837 V=800.0 PL=0
MOVL C00838 V=800.0 PL=0
MOVL C00839 V=800.0 PL=0
MOVL C00840 V=800.0 PL=0
MOVL C00841 V=800.0 PL=0
MOVL C00842 V=800.0 PL=0
MOVL C00843 V=800.0 PL=0
MOVL C00844 V=800.0 PL=0
MOVL C00845 V=800.0 PL=0
MOVL C00846 V=800.0 PL=0
MOVL C00847 V=800.0 PL=0
MOVL C00848 V=800.0 PL=0
MOVL C00849 V=800.0 PL=0
MOVL C00850 V=800.0 PL=0
MOVL C00851 V=800.0 PL=0
MOVL C00852 V=800.0 PL=0
MOVL C00853 V=800.0 PL=0
MOVL C00854 V=800.0 PL=0
MOVL C00855 V=800.0 PL=0
MOVL C00856 V=800.0 PL=0
MOVL C00857 V=800.0 PL=0
MOVL C00858 V=800.0 PL=0
MOVL C00859 V=800.0 PL=0
MOVL C00860 V=800.0 PL=0
MOVL C00861 V=800.0 PL=0
MOVL C00862 V=800.0 PL=0
MOVL C00863 V=800.0 PL=0
MOVL C00864 V=800.0 PL=0
MOVL C00865 V=800.0 PL=0
MOVL C00866 V=800.0 PL=0
MOVL C00867 V=800.0 PL=0
MOVL C00868 V=800.0 PL=0
MOVL C00869 V=800.0 PL=0
MOVL C00870 V=800.0 PL=0
MOVL C00871 V=800.0 PL=0
MOVL C00872 V=800.0 PL=0
MOVL C00873 V=800.0 PL=0
MOVL C00874 V=800.0 PL=0
MOVL C00875 V=800.0 PL=0
MOVL C00876 V=800.0 PL=0
MOVL C00877 V=800.0 PL=0
MOVL C00878 V=800.0 PL=0
MOVL C00879 V=800.0 PL=0
MOVL C00880 V=800.0 PL=0
MOVL C00881 V=800.0 PL=0
MOVL C00882 V=800.0 PL=0
MOVL C00883 V=800.0 PL=0
MOVL C00884 V=800.0 PL=0
MOVL C00885 V=800.0 PL=0
MOVL C00886 V=800.0 PL=0
MOVL C00887 V=800.0 PL=0
MOVL C00888 V=800.0 PL=0
MOVL C00889 V=800.0 PL=0
MOVL C00890 V=800.0 PL=0
MOVL C00891 V=800.0 PL=0
MOVL C00892 V=800.0 PL=0
MOVL C00893 V=800.0 PL=0
MOVL C00894 V=800.0 PL=0
MOVL C00895 V=800.0 PL=0
MOVL C00896 V=800.0 PL=0
MOVL C00897 V=800.0 PL=0
MOVL C00898 V=800.0 PL=0
MOVL C00899 V=800.0 PL=0
MOVL C00900 V=800.0 PL=0
MOVL C00901 V=800.0 PL=0
MOVL C00902 V=800.0 PL=0
MOVL C00903 V=800.0 PL=0
MOVL C00904 V=800.0 PL=0
MOVL C00905 V=800.0 PL=0
MOVL C00906 V=800.0 PL=0
MOVL C00907 V=800.0 PL=0
MOVL C00908 V=800.0 PL=0
MOVL C00909 V=800.0 PL=0
MOVL C00910 V=800.0 PL=0
MOVL C00911 V=800.0 PL=0
MOVL C00912 V=800.0 PL=0
MOVL C00913 V=800.0 PL=0
MOVL C00914 V=800.0 PL=0
MOVL C00915 V=800.0 PL=0
MOVL C00916 V=800.0 PL=0
MOVL C00917 V=800.0 PL=0
MOVL C00918 V=800.0 PL=0
MOVL C00919 V=800.0 PL=0
MOVL C00920 V=800.0 PL=0
MOVL C00921 V=800.0 PL=0
MOVL C00922 V=800.0 PL=0
MOVL C00923 V=800.0 PL=0
MOVL C00924 V=800.0 PL=0
MOVL C00925 V=800.0 PL=0
MOVL C00926 V=800.0 PL=0
MOVL C00927 V=800.0 PL=0
MOVL C00928 V=800.0 PL=0
MOVL C00929 V=800.0 PL=0
MOVL C00930 V=800.0 PL=0
MOVL C00931 V=800.0 PL=0
MOVL C00932 V=800.0 PL=0
MOVL C00933 V=800.0 PL=0
MOVL C00934 V=800.0 PL=0
MOVL C00935 V=800.0 PL=0
MOVL C00936 V=800.0 PL=0
MOVL C00937 V=800.0 PL=0
MOVL C00938 V=800.0 PL=0
MOVL C00939 V=800.0 PL=0
MOVL C00940 V=800.0 PL=0
MOVL C00941 V=800.0 PL=0
MOVL C00942 V=800.0 PL=0
MOVL C00943 V=800.0 PL=0
MOVL C00944 V=800.0 PL=0
MOVL C00945 V=800.0 PL=0
MOVL C00946 V=800.0 PL=0
MOVL C00947 V=800.0 PL=0
MOVL C00948 V=800.0 PL=0
MOVL C00949 V=800.0 PL=0
MOVL C00950 V=800.0 PL=0
MOVL C00951 V=800.0 PL=0
MOVL C00952 V=800.0 PL=0
MOVL C00953 V=800.0 PL=0
MOVL C00954 V=800.0 PL=0
MOVL C00955 V=800.0 PL=0
MOVL C00956 V=800.0 PL=0
MOVL C00957 V=800.0 PL=0
MOVL C00958 V=800.0 PL=0
MOVL C00959 V=800.0 PL=0
MOVL C00960 V=800.0 PL=0
MOVL C00961 V=800.0 PL=0
MOVL C00962 V=800.0 PL=0
MOVL C00963 V=800.0 PL=0
MOVL C00964 V=800.0 PL=0
MOVL C00965 V=800.0 PL=0
MOVL C00966 V=800.0 PL=0
MOVL C00967 V=800.0 PL=0
MOVL C00968 V=800.0 PL=0
MOVL C00969 V=800.0 PL=0
MOVL C00970 V=800.0 PL=0
MOVL C00971 V=800.0 PL=0
MOVL C00972 V=800.0 PL=0
MOVL C00973 V=800.0 PL=0
MOVL C00974 V=800.0 PL=0
MOVL C00975 V=800.0 PL=0
MOVL C00976 V=800.0 PL=0
MOVL C00977 V=800.0 PL=0
MOVL C00978 V=800.0 PL=0
MOVL C00979 V=800.0 PL=0
MOVL C00980 V=800.0 PL=0
MOVL C00981 V=800.0 PL=0
MOVL C00982 V=800.0 PL=0
MOVL C00983 V=800.0 PL=0
MOVL C00984 V=800.0 PL=0
MOVL C00985 V=800.0 PL=0
MOVL C00986 V=800.0 PL=0
MOVL C00987 V=800.0 PL=0
MOVL C00988 V=800.0 PL=0
MOVL C00989 V=800.0 PL=0
MOVL C00990 V=800.0 PL=0
MOVL C00991 V=800.0 PL=0
MOVL C00992 V=800.0 PL=0
MOVL C00993 V=800.0 PL=0
MOVL C00994 V=800.0 PL=0
MOVL C00995 V=800.0 PL=0
MOVL C00996 V=800.0 PL=0
MOVL C00997 V=800.0 PL=0
MOVL C00998 V=800.0 PL=0
MOVL C00999 V=800.0 PL=0
MOVL C01000 V=800.0 PL=0
MOVL C01001 V=800.0 PL=0
MOVL C01002 V=800.0 PL=0
MOVL C01003 V=800.0 PL=0
MOVL C01004 V=800.0 PL=0
MOVL C01005 V=800.0 PL=0
MOVL C01006 V=800.0 PL=0
MOVL C01007 V=800.0 PL=0
MOVL C01008 V=800.0 PL=0
MOVL C01009 V=800.0 PL=0
MOVL C01010 V=800.0 PL=0
MOVL C01011 V=800.0 PL=0
MOVL C01012 V=800.0 PL=0
MOVL C01013 V=800.0 PL=0
MOVL C01014 V=800.0 PL=0
MOVL C01015 V=800.0 PL=0
MOVL C01016 V=800.0 PL=0
MOVL C01017 V=800.0 PL=0
MOVL C01018 V=800.0 PL=0
MOVL C01019 V=800.0 PL=0
MOVL C01020 V=800.0 PL=0
MOVL C01021 V=800.0 PL=0
MOVL C01022 V=800.0 PL=0
MOVL C01023 V=800.0 PL=0
MOVL C01024 V=800.0 PL=0
MOVL C01025 V=800.0 PL=0
MOVL C01026 V=800.0 PL=0
MOVL C01027 V=800.0 PL=0
MOVL C01028 V=800.0 PL=0
MOVL C01029 V=800.0 PL=0
MOVL C01030 V=800.0 PL=0
MOVL C01031 V=800.0 PL=0
MOVL C01032 V=800.0 PL=0
MOVL C01033 V=800.0 PL=0
MOVL C01034 V=800.0 PL=0
MOVL C01035 V=800.0 PL=0
MOVL C01036 V=800.0 PL=0
MOVL C01037 V=800.0 PL=0
MOVL C01038 V=800.0 PL=0
MOVL C01039 V=800.0 PL=0
MOVL C01040 V=800.0 PL=0
MOVL C01041 V=800.0 PL=0
MOVL C01042 V=800.0 PL=0
MOVL C01043 V=800.0 PL=0
MOVL C01044 V=800.0 PL=0
MOVL C01045 V=800.0 PL=0
MOVL C01046 V=800.0 PL=0
MOVL C01047 V=800.0 PL=0
MOVL C01048 V=800.0 PL=0
MOVL C01049 V=800.0 PL=0
MOVL C01050 V=800.0 PL=0
MOVL C01051 V=800.0 PL=0
MOVL C01052 V=800.0 PL=0
MOVL C01053 V=800.0 PL=0
MOVL C01054 V=800.0 PL=0
MOVL C01055 V=800.0 PL=0
MOVL C01056 V=800.0 PL=0
MOVL C01057 V=800.0 PL=0
MOVL C01058 V=800.0 PL=0
MOVL C01059 V=800.0 PL=0
MOVL C01060 V=800.0 PL=0
MOVL C01061 V=800.0 PL=0
MOVL C01062 V=800.0 PL=0
MOVL C01063 V=800.0 PL=0
MOVL C01064 V=800.0 PL=0
MOVL C01065 V=800.0 PL=0
MOVL C01066 V=800.0 PL=0
MOVL C01067 V=800.0 PL=0
MOVL C01068 V=800.0 PL=0
MOVL C01069 V=800.0 PL=0
MOVL C01070 V=800.0 PL=0
MOVL C01071 V=800.0 PL=0
MOVL C01072 V=800.0 PL=0
MOVL C01073 V=800.0 PL=0
MOVL C01074 V=800.0 PL=0
MOVL C01075 V=800.0 PL=0
MOVL C01076 V=800.0 PL=0
MOVL C01077 V=800.0 PL=0
MOVL C01078 V=800.0 PL=0
MOVL C01079 V=800.0 PL=0
MOVL C01080 V=800.0 PL=0
MOVL C01081 V=800.0 PL=0
MOVL C01082 V=800.0 PL=0
MOVL C01083 V=800.0 PL=0
MOVL C01084 V=800.0 PL=0
MOVL C01085 V=800.0 PL=0
MOVL C01086 V=800.0 PL=0
MOVL C01087 V=800.0 PL=0
MOVL C01088 V=800.0 PL=0
MOVL C01089 V=800.0 PL=0
MOVL C01090 V=800.0 PL=0
MOVL C01091 V=800.0 PL=0
MOVL C01092 V=800.0 PL=0
MOVL C01093 V=800.0 PL=0
MOVL C01094 V=800.0 PL=0
MOVL C01095 V=800.0 PL=0
MOVL C01096 V=800.0 PL=0
MOVL C01097 V=800.0 PL=0
MOVL C01098 V=800.0 PL=0
MOVL C01099 V=800.0 PL=0
MOVL C01100 V=800.0 PL=0
MOVL C01101 V=800.0 PL=0
MOVL C01102 V=800.0 PL=0
MOVL C01103 V=800.0 PL=0
MOVL C01104 V=800.0 PL=0
MOVL C01105 V=800.0 PL=0
MOVL C01106 V=800.0 PL=0
MOVL C01107 V=800.0 PL=0
MOVL C01108 V=800.0 PL=0
MOVL C01109 V=800.0 PL=0
MOVL C01110 V=800.0 PL=0
MOVL C01111 V=800.0 PL=0
MOVL C01112 V=800.0 PL=0
MOVL C01113 V=800.0 PL=0
MOVL C01114 V=800.0 PL=0
MOVL C01115 V=800.0 PL=0
MOVL C01116 V=800.0 PL=0
MOVL C01117 V=800.0 PL=0
MOVL C01118 V=800.0 PL=0
MOVL C01119 V=800.0 PL=0
MOVL C01120 V=800.0 PL=0
MOVL C01121 V=800.0 PL=0
MOVL C01122 V=800.0 PL=0
MOVL C01123 V=800.0 PL=0
MOVL C01124 V=800.0 PL=0
MOVL C01125 V=800.0 PL=0
MOVL C01126 V=800.0 PL=0
MOVL C01127 V=800.0 PL=0
MOVL C01128 V=800.0 PL=0
MOVL C01129 V=800.0 PL=0
MOVL C01130 V=800.0 PL=0
MOVL C01131 V=800.0 PL=0
MOVL C01132 V=800.0 PL=0
MOVL C01133 V=800.0 PL=0
MOVL C01134 V=800.0 PL=0
MOVL C01135 V=800.0 PL=0
MOVL C01136 V=800.0 PL=0
MOVL C01137 V=800.0 PL=0
MOVL C01138 V=800.0 PL=0
MOVL C01139 V=800.0 PL=0
MOVL C01140 V=800.0 PL=0
MOVL C01141 V=800.0 PL=0
MOVL C01142 V=800.0 PL=0
MOVL C01143 V=800.0 PL=0
MOVL C01144 V=800.0 PL=0
MOVL C01145 V=800.0 PL=0
MOVL C01146 V=800.0 PL=0
MOVL C01147 V=800.0 PL=0
MOVL C01148 V=800.0 PL=0
MOVL C01149 V=800.0 PL=0
MOVL C01150 V=800.0 PL=0
MOVL C01151 V=800.0 PL=0
MOVL C01152 V=800.0 PL=0
MOVL C01153 V=800.0 PL=0
MOVL C01154 V=800.0 PL=0
MOVL C01155 V=800.0 PL=0
MOVL C01156 V=800.0 PL=0
MOVL C01157 V=800.0 PL=0
MOVL C01158 V=800.0 PL=0
MOVL C01159 V=800.0 PL=0
MOVL C01160 V=800.0 PL=0
MOVL C01161 V=800.0 PL=0
MOVL C01162 V=800.0 PL=0
MOVL C01163 V=800.0 PL=0
MOVL C01164 V=800.0 PL=0
MOVL C01165 V=800.0 PL=0
MOVL C01166 V=800.0 PL=0
MOVL C01167 V=800.0 PL=0
MOVL C01168 V=800.0 PL=0
MOVL C01169 V=800.0 PL=0
MOVL C01170 V=800.0 PL=0
MOVL C01171 V=800.0 PL=0
MOVL C01172 V=800.0 PL=0
MOVL C01173 V=800.0 PL=0
MOVL C01174 V=800.0 PL=0
MOVL C01175 V=800.0 PL=0
MOVL C01176 V=800.0 PL=0
MOVL C01177 V=800.0 PL=0
MOVL C01178 V=800.0 PL=0
MOVL C01179 V=800.0 PL=0
MOVL C01180 V=800.0 PL=0
MOVL C01181 V=800.0 PL=0
MOVL C01182 V=800.0 PL=0
MOVL C01183 V=800.0 PL=0
MOVL C01184 V=800.0 PL=0
MOVL C01185 V=800.0 PL=0
MOVL C01186 V=800.0 PL=0
MOVL C01187 V=800.0 PL=0
MOVL C01188 V=800.0 PL=0
MOVL C01189 V=800.0 PL=0
MOVL C01190 V=800.0 PL=0
MOVL C01191 V=800.0 PL=0
MOVL C01192 V=800.0 PL=0
MOVL C01193 V=800.0 PL=0
MOVL C01194 V=800.0 PL=0
MOVL C01195 V=800.0 PL=0
MOVL C01196 V=800.0 PL=0
MOVL C01197 V=800.0 PL=0
MOVL C01198 V=800.0 PL=0
MOVL C01199 V=800.0 PL=0
MOVL C01200 V=800.0 PL=0
MOVL C01201 V=800.0 PL=0
MOVL C01202 V=800.0 PL=0
MOVL C01203 V=800.0 PL=0
MOVL C01204 V=800.0 PL=0
MOVL C01205 V=800.0 PL=0
MOVL C01206 V=800.0 PL=0
MOVL C01207 V=800.0 PL=0
MOVL C01208 V=800.0 PL=0
MOVL C01209 V=800.0 PL=0
MOVL C01210 V=800.0 PL=0
MOVL C01211 V=800.0 PL=0
MOVL C01212 V=800.0 PL=0
MOVL C01213 V=800.0 PL=0
MOVL C01214 V=800.0 PL=0
MOVL C01215 V=800.0 PL=0
MOVL C01216 V=800.0 PL=0
MOVL C01217 V=800.0 PL=0
MOVL C01218 V=800.0 PL=0
MOVL C01219 V=800.0 PL=0
MOVL C01220 V=800.0 PL=0
MOVL C01221 V=800.0 PL=0
MOVL C01222 V=800.0 PL=0
MOVL C01223 V=800.0 PL=0
MOVL C01224 V=800.0 PL=0
MOVL C01225 V=800.0 PL=0
MOVL C01226 V=800.0 PL=0
MOVL C01227 V=800.0 PL=0
MOVL C01228 V=800.0 PL=0
MOVL C01229 V=800.0 PL=0
MOVL C01230 V=800.0 PL=0
MOVL C01231 V=800.0 PL=0
MOVL C01232 V=800.0 PL=0
MOVL C01233 V=800.0 PL=0
MOVL C01234 V=800.0 PL=0
MOVL C01235 V=800.0 PL=0
MOVL C01236 V=800.0 PL=0
MOVL C01237 V=800.0 PL=0
MOVL C01238 V=800.0 PL=0
MOVL C01239 V=800.0 PL=0
MOVL C01240 V=800.0 PL=0
MOVL C01241 V=800.0 PL=0
MOVL C01242 V=800.0 PL=0
MOVL C01243 V=800.0 PL=0
MOVL C01244 V=800.0 PL=0
MOVL C01245 V=800.0 PL=0
MOVL C01246 V=800.0 PL=0
MOVL C01247 V=800.0 PL=0
MOVL C01248 V=800.0 PL=0
MOVL C01249 V=800.0 PL=0
MOVL C01250 V=800.0 PL=0
MOVL C01251 V=800.0 PL=0
MOVL C01252 V=800.0 PL=0
MOVL C01253 V=800.0 PL=0
MOVL C01254 V=800.0 PL=0
MOVL C01255 V=800.0 PL=0
MOVL C01256 V=800.0 PL=0
MOVL C01257 V=800.0 PL=0
MOVL C01258 V=800.0 PL=0
MOVL C01259 V=800.0 PL=0
MOVL C01260 V=800.0 PL=0
MOVL C01261 V=800.0 PL=0
MOVL C01262 V=800.0 PL=0
MOVL C01263 V=800.0 PL=0
MOVL C01264 V=800.0 PL=0
MOVL C01265 V=800.0 PL=0
MOVL C01266 V=800.0 PL=0
MOVL C01267 V=800.0 PL=0
MOVL C01268 V=800.0 PL=0
MOVL C01269 V=800.0 PL=0
MOVL C01270 V=800.0 PL=0
MOVL C01271 V=800.0 PL=0
MOVL C01272 V=800.0 PL=0
MOVL C01273 V=800.0 PL=0
MOVL C01274 V=800.0 PL=0
MOVL C01275 V=800.0 PL=0
MOVL C01276 V=800.0 PL=0
MOVL C01277 V=800.0 PL=0
MOVL C01278 V=800.0 PL=0
MOVL C01279 V=800.0 PL=0
MOVL C01280 V=800.0 PL=0
MOVL C01281 V=800.0 PL=0
MOVL C01282 V=800.0 PL=0
MOVL C01283 V=800.0 PL=0
MOVL C01284 V=800.0 PL=0
MOVL C01285 V=800.0 PL=0
MOVL C01286 V=800.0 PL=0
MOVL C01287 V=800.0 PL=0
MOVL C01288 V=800.0 PL=0
MOVL C01289 V=800.0 PL=0
MOVL C01290 V=800.0 PL=0
MOVL C01291 V=800.0 PL=0
MOVL C01292 V=800.0 PL=0
MOVL C01293 V=800.0 PL=0
MOVL C01294 V=800.0 PL=0
MOVL C01295 V=800.0 PL=0
MOVL C01296 V=800.0 PL=0
MOVL C01297 V=800.0 PL=0
MOVL C01298 V=800.0 PL=0
MOVL C01299 V=800.0 PL=0
MOVL C01300 V=800.0 PL=0
MOVL C01301 V=800.0 PL=0
MOVL C01302 V=800.0 PL=0
MOVL C01303 V=800.0 PL=0
MOVL C01304 V=800.0 PL=0
MOVL C01305 V=800.0 PL=0
MOVL C01306 V=800.0 PL=0
MOVL C01307 V=800.0 PL=0
MOVL C01308 V=800.0 PL=0
MOVL C01309 V=800.0 PL=0
MOVL C01310 V=800.0 PL=0
MOVL C01311 V=800.0 PL=0
MOVL C01312 V=800.0 PL=0
MOVL C01313 V=800.0 PL=0
MOVL C01314 V=800.0 PL=0
MOVL C01315 V=800.0 PL=0
MOVL C01316 V=800.0 PL=0
MOVL C01317 V=800.0 PL=0
MOVL C01318 V=800.0 PL=0
MOVL C01319 V=800.0 PL=0
MOVL C01320 V=800.0 PL=0
MOVL C01321 V=800.0 PL=0
MOVL C01322 V=800.0 PL=0
MOVL C01323 V=800.0 PL=0
MOVL C01324 V=800.0 PL=0
MOVL C01325 V=800.0 PL=0
MOVL C01326 V=800.0 PL=0
MOVL C01327 V=800.0 PL=0
MOVL C01328 V=800.0 PL=0
MOVL C01329 V=800.0 PL=0
MOVL C01330 V=800.0 PL=0
MOVL C01331 V=800.0 PL=0
MOVL C01332 V=800.0 PL=0
MOVL C01333 V=800.0 PL=0
MOVL C01334 V=800.0 PL=0
MOVL C01335 V=800.0 PL=0
MOVL C01336 V=800.0 PL=0
MOVL C01337 V=800.0 PL=0
MOVL C01338 V=800.0 PL=0
MOVL C01339 V=800.0 PL=0
MOVL C01340 V=800.0 PL=0
MOVL C01341 V=800.0 PL=0
MOVL C01342 V=800.0 PL=0
MOVL C01343 V=800.0 PL=0
MOVL C01344 V=800.0 PL=0
MOVL C01345 V=800.0 PL=0
MOVL C01346 V=800.0 PL=0
MOVL C01347 V=800.0 PL=0
MOVL C01348 V=800.0 PL=0
MOVL C01349 V=800.0 PL=0
MOVL C01350 V=800.0 PL=0
MOVL C01351 V=800.0 PL=0
MOVL C01352 V=800.0 PL=0
MOVL C01353 V=800.0 PL=0
MOVL C01354 V=800.0 PL=0
MOVL C01355 V=800.0 PL=0
MOVL C01356 V=800.0 PL=0
MOVL C01357 V=800.0 PL=0
MOVL C01358 V=800.0 PL=0
MOVL C01359 V=800.0 PL=0
MOVL C01360 V=800.0 PL=0
MOVL C01361 V=800.0 PL=0
MOVL C01362 V=800.0 PL=0
MOVL C01363 V=800.0 PL=0
MOVL C01364 V=800.0 PL=0
MOVL C01365 V=800.0 PL=0
MOVL C01366 V=800.0 PL=0
MOVL C01367 V=800.0 PL=0
MOVL C01368 V=800.0 PL=0
MOVL C01369 V=800.0 PL=0
MOVL C01370 V=800.0 PL=0
MOVL C01371 V=800.0 PL=0
MOVL C01372 V=800.0 PL=0
MOVL C01373 V=800.0 PL=0
MOVL C01374 V=800.0 PL=0
MOVL C01375 V=800.0 PL=0
MOVL C01376 V=800.0 PL=0
MOVL C01377 V=800.0 PL=0
MOVL C01378 V=800.0 PL=0
MOVL C01379 V=800.0 PL=0
MOVL C01380 V=800.0 PL=0
MOVL C01381 V=800.0 PL=0
MOVL C01382 V=800.0 PL=0
MOVL C01383 V=800.0 PL=0
MOVL C01384 V=800.0 PL=0
MOVL C01385 V=800.0 PL=0
MOVL C01386 V=800.0 PL=0
MOVL C01387 V=800.0 PL=0
MOVL C01388 V=800.0 PL=0
MOVL C01389 V=800.0 PL=0
MOVL C01390 V=800.0 PL=0
MOVL C01391 V=800.0 PL=0
MOVL C01392 V=800.0 PL=0
MOVL C01393 V=800.0 PL=0
MOVL C01394 V=800.0 PL=0
MOVL C01395 V=800.0 PL=0
MOVL C01396 V=800.0 PL=0
MOVL C01397 V=800.0 PL=0
MOVL C01398 V=800.0 PL=0
MOVL C01399 V=800.0 PL=0
MOVL C01400 V=800.0 PL=0
MOVL C01401 V=800.0 PL=0
MOVL C01402 V=800.0 PL=0
MOVL C01403 V=800.0 PL=0
MOVL C01404 V=800.0 PL=0
MOVL C01405 V=800.0 PL=0
MOVL C01406 V=800.0 PL=0
MOVL C01407 V=800.0 PL=0
MOVL C01408 V=800.0 PL=0
MOVL C01409 V=800.0 PL=0
MOVL C01410 V=800.0 PL=0
MOVL C01411 V=800.0 PL=0
MOVL C01412 V=800.0 PL=0
MOVL C01413 V=800.0 PL=0
MOVL C01414 V=800.0 PL=0
MOVL C01415 V=800.0 PL=0
MOVL C01416 V=800.0 PL=0
MOVL C01417 V=800.0 PL=0
MOVL C01418 V=800.0 PL=0
MOVL C01419 V=800.0 PL=0
MOVL C01420 V=800.0 PL=0
MOVL C01421 V=800.0 PL=0
MOVL C01422 V=800.0 PL=0
MOVL C01423 V=800.0 PL=0
MOVL C01424 V=800.0 PL=0
MOVL C01425 V=800.0 PL=0
MOVL C01426 V=800.0 PL=0
MOVL C01427 V=800.0 PL=0
MOVL C01428 V=800.0 PL=0
MOVL C01429 V=800.0 PL=0
MOVL C01430 V=800.0 PL=0
MOVL C01431 V=800.0 PL=0
MOVL C01432 V=800.0 PL=0
MOVL C01433 V=800.0 PL=0
MOVL C01434 V=800.0 PL=0
MOVL C01435 V=800.0 PL=0
MOVL C01436 V=800.0 PL=0
MOVL C01437 V=800.0 PL=0
MOVL C01438 V=800.0 PL=0
MOVL C01439 V=800.0 PL=0
MOVL C01440 V=800.0 PL=0
MOVL C01441 V=800.0 PL=0
MOVL C01442 V=800.0 PL=0
MOVL C01443 V=800.0 PL=0
MOVL C01444 V=800.0 PL=0
MOVL C01445 V=800.0 PL=0
MOVL C01446 V=800.0 PL=0
MOVL C01447 V=800.0 PL=0
MOVL C01448 V=800.0 PL=0
MOVL C01449 V=800.0 PL=0
MOVL C01450 V=800.0 PL=0
MOVL C01451 V=800.0 PL=0
MOVL C01452 V=800.0 PL=0
MOVL C01453 V=800.0 PL=0
MOVL C01454 V=800.0 PL=0
MOVL C01455 V=800.0 PL=0
MOVL C01456 V=800.0 PL=0
MOVL C01457 V=800.0 PL=0
MOVL C01458 V=800.0 PL=0
MOVL C01459 V=800.0 PL=0
MOVL C01460 V=800.0 PL=0
MOVL C01461 V=800.0 PL=0
MOVL C01462 V=800.0 PL=0
MOVL C01463 V=800.0 PL=0
MOVL C01464 V=800.0 PL=0
MOVL C01465 V=800.0 PL=0
MOVL C01466 V=800.0 PL=0
MOVL C01467 V=800.0 PL=0
MOVL C01468 V=800.0 PL=0
MOVL C01469 V=800.0 PL=0
MOVL C01470 V=800.0 PL=0
MOVL C01471 V=800.0 PL=0
MOVL C01472 V=800.0 PL=0
MOVL C01473 V=800.0 PL=0
MOVL C01474 V=800.0 PL=0
MOVL C01475 V=800.0 PL=0
MOVL C01476 V=800.0 PL=0
MOVL C01477 V=800.0 PL=0
MOVL C01478 V=800.0 PL=0
MOVL C01479 V=800.0 PL=0
MOVL C01480 V=800.0 PL=0
MOVL C01481 V=800.0 PL=0
MOVL C01482 V=800.0 PL=0
MOVL C01483 V=800.0 PL=0
MOVL C01484 V=800.0 PL=0
MOVL C01485 V=800.0 PL=0
MOVL C01486 V=800.0 PL=0
MOVL C01487 V=800.0 PL=0
MOVL C01488 V=800.0 PL=0
MOVL C01489 V=800.0 PL=0
MOVL C01490 V=800.0 PL=0
MOVL C01491 V=800.0 PL=0
MOVL C01492 V=800.0 PL=0
MOVL C01493 V=800.0 PL=0
MOVL C01494 V=800.0 PL=0
MOVL C01495 V=800.0 PL=0
MOVL C01496 V=800.0 PL=0
MOVL C01497 V=800.0 PL=0
MOVL C01498 V=800.0 PL=0
MOVL C01499 V=800.0 PL=0
MOVL C01500 V=800.0 PL=0
MOVL C01501 V=800.0 PL=0
MOVL C01502 V=800.0 PL=0
MOVL C01503 V=800.0 PL=0
MOVL C01504 V=800.0 PL=0
MOVL C01505 V=800.0 PL=0
MOVL C01506 V=800.0 PL=0
MOVL C01507 V=800.0 PL=0
MOVL C01508 V=800.0 PL=0
MOVL C01509 V=800.0 PL=0
MOVL C01510 V=800.0 PL=0
MOVL C01511 V=800.0 PL=0
MOVL C01512 V=800.0 PL=0
MOVL C01513 V=800.0 PL=0
MOVL C01514 V=800.0 PL=0
MOVL C01515 V=800.0 PL=0
MOVL C01516 V=800.0 PL=0
MOVL C01517 V=800.0 PL=0
MOVL C01518 V=800.0 PL=0
MOVL C01519 V=800.0 PL=0
MOVL C01520 V=800.0 PL=0
MOVL C01521 V=800.0 PL=0
MOVL C01522 V=800.0 PL=0
MOVL C01523 V=800.0 PL=0
MOVL C01524 V=800.0 PL=0
MOVL C01525 V=800.0 PL=0
MOVL C01526 V=800.0 PL=0
MOVL C01527 V=800.0 PL=0
MOVL C01528 V=800.0 PL=0
MOVL C01529 V=800.0 PL=0
MOVL C01530 V=800.0 PL=0
MOVL C01531 V=800.0 PL=0
MOVL C01532 V=800.0 PL=0
MOVL C01533 V=800.0 PL=0
MOVL C01534 V=800.0 PL=0
MOVL C01535 V=800.0 PL=0
MOVL C01536 V=800.0 PL=0
MOVL C01537 V=800.0 PL=0
MOVL C01538 V=800.0 PL=0
MOVL C01539 V=800.0 PL=0
MOVL C01540 V=800.0 PL=0
MOVL C01541 V=800.0 PL=0
MOVL C01542 V=800.0 PL=0
MOVL C01543 V=800.0 PL=0
MOVL C01544 V=800.0 PL=0
MOVL C01545 V=800.0 PL=0
MOVL C01546 V=800.0 PL=0
MOVL C01547 V=800.0 PL=0
MOVL C01548 V=800.0 PL=0
MOVL C01549 V=800.0 PL=0
MOVL C01550 V=800.0 PL=0
MOVL C01551 V=800.0 PL=0
MOVL C01552 V=800.0 PL=0
MOVL C01553 V=800.0 PL=0
MOVL C01554 V=800.0 PL=0
MOVL C01555 V=800.0 PL=0
MOVL C01556 V=800.0 PL=0
MOVL C01557 V=800.0 PL=0
MOVL C01558 V=800.0 PL=0
MOVL C01559 V=800.0 PL=0
MOVL C01560 V=800.0 PL=0
MOVL C01561 V=800.0 PL=0
MOVL C01562 V=800.0 PL=0
MOVL C01563 V=800.0 PL=0
MOVL C01564 V=800.0 PL=0
MOVL C01565 V=800.0 PL=0
MOVL C01566 V=800.0 PL=0
MOVL C01567 V=800.0 PL=0
MOVL C01568 V=800.0 PL=0
MOVL C01569 V=800.0 PL=0
MOVL C01570 V=800.0 PL=0
MOVL C01571 V=800.0 PL=0
MOVL C01572 V=800.0 PL=0
MOVL C01573 V=800.0 PL=0
MOVL C01574 V=800.0 PL=0
MOVL C01575 V=800.0 PL=0
MOVL C01576 V=800.0 PL=0
MOVL C01577 V=800.0 PL=0
MOVL C01578 V=800.0 PL=0
MOVL C01579 V=800.0 PL=0
MOVL C01580 V=800.0 PL=0
MOVL C01581 V=800.0 PL=0
MOVL C01582 V=800.0 PL=0
MOVL C01583 V=800.0 PL=0
MOVL C01584 V=800.0 PL=0
MOVL C01585 V=800.0 PL=0
MOVL C01586 V=800.0 PL=0
MOVL C01587 V=800.0 PL=0
MOVL C01588 V=800.0 PL=0
MOVL C01589 V=800.0 PL=0
MOVL C01590 V=800.0 PL=0
MOVL C01591 V=800.0 PL=0
MOVL C01592 V=800.0 PL=0
MOVL C01593 V=800.0 PL=0
MOVL C01594 V=800.0 PL=0
MOVL C01595 V=800.0 PL=0
MOVL C01596 V=800.0 PL=0
MOVL C01597 V=800.0 PL=0
MOVL C01598 V=800.0 PL=0
MOVL C01599 V=800.0 PL=0
MOVL C01600 V=800.0 PL=0
MOVL C01601 V=800.0 PL=0
MOVL C01602 V=800.0 PL=0
MOVL C01603 V=800.0 PL=0
MOVL C01604 V=800.0 PL=0
MOVL C01605 V=800.0 PL=0
MOVL C01606 V=800.0 PL=0
MOVL C01607 V=800.0 PL=0
MOVL C01608 V=800.0 PL=0
MOVL C01609 V=800.0 PL=0
MOVL C01610 V=800.0 PL=0
MOVL C01611 V=800.0 PL=0
MOVL C01612 V=800.0 PL=0
MOVL C01613 V=800.0 PL=0
MOVL C01614 V=800.0 PL=0
MOVL C01615 V=800.0 PL=0
MOVL C01616 V=800.0 PL=0
MOVL C01617 V=800.0 PL=0
MOVL C01618 V=800.0 PL=0
MOVL C01619 V=800.0 PL=0
MOVL C01620 V=800.0 PL=0
MOVL C01621 V=800.0 PL=0
MOVL C01622 V=800.0 PL=0
MOVL C01623 V=800.0 PL=0
MOVL C01624 V=800.0 PL=0
MOVL C01625 V=800.0 PL=0
MOVL C01626 V=800.0 PL=0
MOVL C01627 V=800.0 PL=0
MOVL C01628 V=800.0 PL=0
MOVL C01629 V=800.0 PL=0
MOVL C01630 V=800.0 PL=0
MOVL C01631 V=800.0 PL=0
MOVL C01632 V=800.0 PL=0
MOVL C01633 V=800.0 PL=0
MOVL C01634 V=800.0 PL=0
MOVL C01635 V=800.0 PL=0
MOVL C01636 V=800.0 PL=0
MOVL C01637 V=800.0 PL=0
MOVL C01638 V=800.0 PL=0
MOVL C01639 V=800.0 PL=0
MOVL C01640 V=800.0 PL=0
MOVL C01641 V=800.0 PL=0
MOVL C01642 V=800.0 PL=0
MOVL C01643 V=800.0 PL=0
MOVL C01644 V=800.0 PL=0
MOVL C01645 V=800.0 PL=0
MOVL C01646 V=800.0 PL=0
MOVL C01647 V=800.0 PL=0
MOVL C01648 V=800.0 PL=0
MOVL C01649 V=800.0 PL=0
MOVL C01650 V=800.0 PL=0
MOVL C01651 V=800.0 PL=0
MOVL C01652 V=800.0 PL=0
MOVL C01653 V=800.0 PL=0
MOVL C01654 V=800.0 PL=0
MOVL C01655 V=800.0 PL=0
MOVL C01656 V=800.0 PL=0
MOVL C01657 V=800.0 PL=0
MOVL C01658 V=800.0 PL=0
MOVL C01659 V=800.0 PL=0
MOVL C01660 V=800.0 PL=0
MOVL C01661 V=800.0 PL=0
MOVL C01662 V=800.0 PL=0
MOVL C01663 V=800.0 PL=0
MOVL C01664 V=800.0 PL=0
MOVL C01665 V=800.0 PL=0
MOVL C01666 V=800.0 PL=0
MOVL C01667 V=800.0 PL=0
MOVL C01668 V=800.0 PL=0
MOVL C01669 V=800.0 PL=0
MOVL C01670 V=800.0 PL=0
MOVL C01671 V=800.0 PL=0
MOVL C01672 V=800.0 PL=0
MOVL C01673 V=800.0 PL=0
MOVL C01674 V=800.0 PL=0
MOVL C01675 V=800.0 PL=0
MOVL C01676 V=800.0 PL=0
MOVL C01677 V=800.0 PL=0
MOVL C01678 V=800.0 PL=0
MOVL C01679 V=800.0 PL=0
MOVL C01680 V=800.0 PL=0
MOVL C01681 V=800.0 PL=0
MOVL C01682 V=800.0 PL=0
MOVL C01683 V=800.0 PL=0
MOVL C01684 V=800.0 PL=0
MOVL C01685 V=800.0 PL=0
MOVL C01686 V=800.0 PL=0
MOVL C01687 V=800.0 PL=0
MOVL C01688 V=800.0 PL=0
MOVL C01689 V=800.0 PL=0
MOVL C01690 V=800.0 PL=0
MOVL C01691 V=800.0 PL=0
MOVL C01692 V=800.0 PL=0
MOVL C01693 V=800.0 PL=0
MOVL C01694 V=800.0 PL=0
MOVL C01695 V=800.0 PL=0
MOVL C01696 V=800.0 PL=0
MOVL C01697 V=800.0 PL=0
MOVL C01698 V=800.0 PL=0
MOVL C01699 V=800.0 PL=0
MOVL C01700 V=800.0 PL=0
MOVL C01701 V=800.0 PL=0
MOVL C01702 V=800.0 PL=0
MOVL C01703 V=800.0 PL=0
MOVL C01704 V=800.0 PL=0
MOVL C01705 V=800.0 PL=0
MOVL C01706 V=800.0 PL=0
MOVL C01707 V=800.0 PL=0
MOVL C01708 V=800.0 PL=0
MOVL C01709 V=800.0 PL=0
MOVL C01710 V=800.0 PL=0
MOVL C01711 V=800.0 PL=0
MOVL C01712 V=800.0 PL=0
MOVL C01713 V=800.0 PL=0
MOVL C01714 V=800.0 PL=0
MOVL C01715 V=800.0 PL=0
MOVL C01716 V=800.0 PL=0
MOVL C01717 V=800.0 PL=0
MOVL C01718 V=800.0 PL=0
MOVL C01719 V=800.0 PL=0
MOVL C01720 V=800.0 PL=0
MOVL C01721 V=800.0 PL=0
MOVL C01722 V=800.0 PL=0
MOVL C01723 V=800.0 PL=0
MOVL C01724 V=800.0 PL=0
MOVL C01725 V=800.0 PL=0
MOVL C01726 V=800.0 PL=0
MOVL C01727 V=800.0 PL=0
MOVL C01728 V=800.0 PL=0
MOVL C01729 V=800.0 PL=0
MOVL C01730 V=800.0 PL=0
MOVL C01731 V=800.0 PL=0
MOVL C01732 V=800.0 PL=0
MOVL C01733 V=800.0 PL=0
MOVL C01734 V=800.0 PL=0
MOVL C01735 V=800.0 PL=0
MOVL C01736 V=800.0 PL=0
MOVL C01737 V=800.0 PL=0
MOVL C01738 V=800.0 PL=0
MOVL C01739 V=800.0 PL=0
MOVL C01740 V=800.0 PL=0
MOVL C01741 V=800.0 PL=0
MOVL C01742 V=800.0 PL=0
MOVL C01743 V=800.0 PL=0
MOVL C01744 V=800.0 PL=0
MOVL C01745 V=800.0 PL=0
MOVL C01746 V=800.0 PL=0
MOVL C01747 V=800.0 PL=0
MOVL C01748 V=800.0 PL=0
MOVL C01749 V=800.0 PL=0
MOVL C01750 V=800.0 PL=0
MOVL C01751 V=800.0 PL=0
MOVL C01752 V=800.0 PL=0
MOVL C01753 V=800.0 PL=0
MOVL C01754 V=800.0 PL=0
MOVL C01755 V=800.0 PL=0
MOVL C01756 V=800.0 PL=0
MOVL C01757 V=800.0 PL=0
MOVL C01758 V=800.0 PL=0
MOVL C01759 V=800.0 PL=0
MOVL C01760 V=800.0 PL=0
MOVL C01761 V=800.0 PL=0
MOVL C01762 V=800.0 PL=0
MOVL C01763 V=800.0 PL=0
MOVL C01764 V=800.0 PL=0
MOVL C01765 V=800.0 PL=0
MOVL C01766 V=800.0 PL=0
MOVL C01767 V=800.0 PL=0
MOVL C01768 V=800.0 PL=0
MOVL C01769 V=800.0 PL=0
MOVL C01770 V=800.0 PL=0
MOVL C01771 V=800.0 PL=0
MOVL C01772 V=800.0 PL=0
MOVL C01773 V=800.0 PL=0
MOVL C01774 V=800.0 PL=0
MOVL C01775 V=800.0 PL=0
MOVL C01776 V=800.0 PL=0
MOVL C01777 V=800.0 PL=0
MOVL C01778 V=800.0 PL=0
MOVL C01779 V=800.0 PL=0
MOVL C01780 V=800.0 PL=0
MOVL C01781 V=800.0 PL=0
MOVL C01782 V=800.0 PL=0
MOVL C01783 V=800.0 PL=0
MOVL C01784 V=800.0 PL=0
MOVL C01785 V=800.0 PL=0
MOVL C01786 V=800.0 PL=0
MOVL C01787 V=800.0 PL=0
MOVL C01788 V=800.0 PL=0
MOVL C01789 V=800.0 PL=0
MOVL C01790 V=800.0 PL=0
MOVL C01791 V=800.0 PL=0
MOVL C01792 V=800.0 PL=0
MOVL C01793 V=800.0 PL=0
MOVL C01794 V=800.0 PL=0
MOVL C01795 V=800.0 PL=0
MOVL C01796 V=800.0 PL=0
MOVL C01797 V=800.0 PL=0
MOVL C01798 V=800.0 PL=0
MOVL C01799 V=800.0 PL=0
MOVL C01800 V=800.0 PL=0
MOVL C01801 V=800.0 PL=0
MOVL C01802 V=800.0 PL=0
MOVL C01803 V=800.0 PL=0
MOVL C01804 V=800.0 PL=0
MOVL C01805 V=800.0 PL=0
MOVL C01806 V=800.0 PL=0
MOVL C01807 V=800.0 PL=0
MOVL C01808 V=800.0 PL=0
MOVL C01809 V=800.0 PL=0
MOVL C01810 V=800.0 PL=0
MOVL C01811 V=800.0 PL=0
MOVL C01812 V=800.0 PL=0
MOVL C01813 V=800.0 PL=0
MOVL C01814 V=800.0 PL=0
MOVL C01815 V=800.0 PL=0
MOVL C01816 V=800.0 PL=0
MOVL C01817 V=800.0 PL=0
MOVL C01818 V=800.0 PL=0
MOVL C01819 V=800.0 PL=0
MOVL C01820 V=800.0 PL=0
MOVL C01821 V=800.0 PL=0
MOVL C01822 V=800.0 PL=0
MOVL C01823 V=800.0 PL=0
MOVL C01824 V=800.0 PL=0
MOVL C01825 V=800.0 PL=0
MOVL C01826 V=800.0 PL=0
MOVL C01827 V=800.0 PL=0
MOVL C01828 V=800.0 PL=0
MOVL C01829 V=800.0 PL=0
MOVL C01830 V=800.0 PL=0
MOVL C01831 V=800.0 PL=0
MOVL C01832 V=800.0 PL=0
MOVL C01833 V=800.0 PL=0
MOVL C01834 V=800.0 PL=0
MOVL C01835 V=800.0 PL=0
MOVL C01836 V=800.0 PL=0
MOVL C01837 V=800.0 PL=0
MOVL C01838 V=800.0 PL=0
MOVL C01839 V=800.0 PL=0
MOVL C01840 V=800.0 PL=0
MOVL C01841 V=800.0 PL=0
MOVL C01842 V=800.0 PL=0
MOVL C01843 V=800.0 PL=0
MOVL C01844 V=800.0 PL=0
MOVL C01845 V=800.0 PL=0
MOVL C01846 V=800.0 PL=0
MOVL C01847 V=800.0 PL=0
MOVL C01848 V=800.0 PL=0
MOVL C01849 V=800.0 PL=0
MOVL C01850 V=800.0 PL=0
MOVL C01851 V=800.0 PL=0
MOVL C01852 V=800.0 PL=0
MOVL C01853 V=800.0 PL=0
MOVL C01854 V=800.0 PL=0
MOVL C01855 V=800.0 PL=0
MOVL C01856 V=800.0 PL=0
MOVL C01857 V=800.0 PL=0
MOVL C01858 V=800.0 PL=0
MOVL C01859 V=800.0 PL=0
MOVL C01860 V=800.0 PL=0
MOVL C01861 V=800.0 PL=0
MOVL C01862 V=800.0 PL=0
MOVL C01863 V=800.0 PL=0
MOVL C01864 V=800.0 PL=0
MOVL C01865 V=800.0 PL=0
MOVL C01866 V=800.0 PL=0
MOVL C01867 V=800.0 PL=0
MOVL C01868 V=800.0 PL=0
MOVL C01869 V=800.0 PL=0
MOVL C01870 V=800.0 PL=0
MOVL C01871 V=800.0 PL=0
MOVL C01872 V=800.0 PL=0
MOVL C01873 V=800.0 PL=0
MOVL C01874 V=800.0 PL=0
MOVL C01875 V=800.0 PL=0
MOVL C01876 V=800.0 PL=0
MOVL C01877 V=800.0 PL=0
MOVL C01878 V=800.0 PL=0
MOVL C01879 V=800.0 PL=0
MOVL C01880 V=800.0 PL=0
MOVL C01881 V=800.0 PL=0
MOVL C01882 V=800.0 PL=0
MOVL C01883 V=800.0 PL=0
MOVL C01884 V=800.0 PL=0
MOVL C01885 V=800.0 PL=0
MOVL C01886 V=800.0 PL=0
MOVL C01887 V=800.0 PL=0
MOVL C01888 V=800.0 PL=0
MOVL C01889 V=800.0 PL=0
MOVL C01890 V=800.0 PL=0
MOVL C01891 V=800.0 PL=0
MOVL C01892 V=800.0 PL=0
MOVL C01893 V=800.0 PL=0
MOVL C01894 V=800.0 PL=0
MOVL C01895 V=800.0 PL=0
MOVL C01896 V=800.0 PL=0
MOVL C01897 V=800.0 PL=0
MOVL C01898 V=800.0 PL=0
MOVL C01899 V=800.0 PL=0
MOVL C01900 V=800.0 PL=0
MOVL C01901 V=800.0 PL=0
MOVL C01902 V=800.0 PL=0
MOVL C01903 V=800.0 PL=0
MOVL C01904 V=800.0 PL=0
MOVL C01905 V=800.0 PL=0
MOVL C01906 V=800.0 PL=0
MOVL C01907 V=800.0 PL=0
MOVL C01908 V=800.0 PL=0
MOVL C01909 V=800.0 PL=0
MOVL C01910 V=800.0 PL=0
MOVL C01911 V=800.0 PL=0
MOVL C01912 V=800.0 PL=0
MOVL C01913 V=800.0 PL=0
MOVL C01914 V=800.0 PL=0
MOVL C01915 V=800.0 PL=0
MOVL C01916 V=800.0 PL=0
MOVL C01917 V=800.0 PL=0
MOVL C01918 V=800.0 PL=0
MOVL C01919 V=800.0 PL=0
MOVL C01920 V=800.0 PL=0
MOVL C01921 V=800.0 PL=0
MOVL C01922 V=800.0 PL=0
MOVL C01923 V=800.0 PL=0
MOVL C01924 V=800.0 PL=0
MOVL C01925 V=800.0 PL=0
MOVL C01926 V=800.0 PL=0
MOVL C01927 V=800.0 PL=0
MOVL C01928 V=800.0 PL=0
MOVL C01929 V=800.0 PL=0
MOVL C01930 V=800.0 PL=0
MOVL C01931 V=800.0 PL=0
MOVL C01932 V=800.0 PL=0
MOVL C01933 V=800.0 PL=0
MOVL C01934 V=800.0 PL=0
MOVL C01935 V=800.0 PL=0
MOVL C01936 V=800.0 PL=0
MOVL C01937 V=800.0 PL=0
MOVL C01938 V=800.0 PL=0
MOVL C01939 V=800.0 PL=0
MOVL C01940 V=800.0 PL=0
MOVL C01941 V=800.0 PL=0
MOVL C01942 V=800.0 PL=0
MOVL C01943 V=800.0 PL=0
MOVL C01944 V=800.0 PL=0
MOVL C01945 V=800.0 PL=0
MOVL C01946 V=800.0 PL=0
MOVL C01947 V=800.0 PL=0
MOVL C01948 V=800.0 PL=0
MOVL C01949 V=800.0 PL=0
MOVL C01950 V=800.0 PL=0
MOVL C01951 V=800.0 PL=0
MOVL C01952 V=800.0 PL=0
MOVL C01953 V=800.0 PL=0
MOVL C01954 V=800.0 PL=0
MOVL C01955 V=800.0 PL=0
MOVL C01956 V=800.0 PL=0
MOVL C01957 V=800.0 PL=0
MOVL C01958 V=800.0 PL=0
MOVL C01959 V=800.0 PL=0
MOVL C01960 V=800.0 PL=0
MOVL C01961 V=800.0 PL=0
MOVL C01962 V=800.0 PL=0
MOVL C01963 V=800.0 PL=0
MOVL C01964 V=800.0 PL=0
MOVL C01965 V=800.0 PL=0
MOVL C01966 V=800.0 PL=0
MOVL C01967 V=800.0 PL=0
MOVL C01968 V=800.0 PL=0
MOVL C01969 V=800.0 PL=0
MOVL C01970 V=800.0 PL=0
MOVL C01971 V=800.0 PL=0
MOVL C01972 V=800.0 PL=0
MOVL C01973 V=800.0 PL=0
MOVL C01974 V=800.0 PL=0
MOVL C01975 V=800.0 PL=0
MOVL C01976 V=800.0 PL=0
MOVL C01977 V=800.0 PL=0
MOVL C01978 V=800.0 PL=0
MOVL C01979 V=800.0 PL=0
MOVL C01980 V=800.0 PL=0
MOVL C01981 V=800.0 PL=0
MOVL C01982 V=800.0 PL=0
MOVL C01983 V=800.0 PL=0
MOVL C01984 V=800.0 PL=0
MOVL C01985 V=800.0 PL=0
MOVL C01986 V=800.0 PL=0
MOVL C01987 V=800.0 PL=0
MOVL C01988 V=800.0 PL=0
MOVL C01989 V=800.0 PL=0
MOVL C01990 V=800.0 PL=0
MOVL C01991 V=800.0 PL=0
MOVL C01992 V=800.0 PL=0
MOVL C01993 V=800.0 PL=0
MOVL C01994 V=800.0 PL=0
MOVL C01995 V=800.0 PL=0
MOVL C01996 V=800.0 PL=0
MOVL C01997 V=800.0 PL=0
MOVL C01998 V=800.0 PL=0
MOVL C01999 V=800.0 PL=0
MOVL C02000 V=800.0 PL=0
MOVL C02001 V=800.0 PL=0
MOVL C02002 V=800.0 PL=0
MOVL C02003 V=800.0 PL=0
MOVL C02004 V=800.0 PL=0
MOVL C02005 V=800.0 PL=0
MOVL C02006 V=800.0 PL=0
MOVL C02007 V=800.0 PL=0
MOVL C02008 V=800.0 PL=0
MOVL C02009 V=800.0 PL=0
MOVL C02010 V=800.0 PL=0
MOVL C02011 V=800.0 PL=0
MOVL C02012 V=800.0 PL=0
MOVL C02013 V=800.0 PL=0
MOVL C02014 V=800.0 PL=0
MOVL C02015 V=800.0 PL=0
MOVL C02016 V=800.0 PL=0
MOVL C02017 V=800.0 PL=0
MOVL C02018 V=800.0 PL=0
MOVL C02019 V=800.0 PL=0
MOVL C02020 V=800.0 PL=0
MOVL C02021 V=800.0 PL=0
MOVL C02022 V=800.0 PL=0
MOVL C02023 V=800.0 PL=0
MOVL C02024 V=800.0 PL=0
MOVL C02025 V=800.0 PL=0
MOVL C02026 V=800.0 PL=0
MOVL C02027 V=800.0 PL=0
MOVL C02028 V=800.0 PL=0
MOVL C02029 V=800.0 PL=0
MOVL C02030 V=800.0 PL=0
MOVL C02031 V=800.0 PL=0
MOVL C02032 V=800.0 PL=0
MOVL C02033 V=800.0 PL=0
MOVL C02034 V=800.0 PL=0
MOVL C02035 V=800.0 PL=0
MOVL C02036 V=800.0 PL=0
MOVL C02037 V=800.0 PL=0
MOVL C02038 V=800.0 PL=0
MOVL C02039 V=800.0 PL=0
MOVL C02040 V=800.0 PL=0
MOVL C02041 V=800.0 PL=0
MOVL C02042 V=800.0 PL=0
MOVL C02043 V=800.0 PL=0
MOVL C02044 V=800.0 PL=0
MOVL C02045 V=800.0 PL=0
MOVL C02046 V=800.0 PL=0
MOVL C02047 V=800.0 PL=0
MOVL C02048 V=800.0 PL=0
MOVL C02049 V=800.0 PL=0
MOVL C02050 V=800.0 PL=0
MOVL C02051 V=800.0 PL=0
MOVL C02052 V=800.0 PL=0
MOVL C02053 V=800.0 PL=0
MOVL C02054 V=800.0 PL=0
MOVL C02055 V=800.0 PL=0
MOVL C02056 V=800.0 PL=0
MOVL C02057 V=800.0 PL=0
MOVL C02058 V=800.0 PL=0
MOVL C02059 V=800.0 PL=0
MOVL C02060 V=800.0 PL=0
MOVL C02061 V=800.0 PL=0
MOVL C02062 V=800.0 PL=0
MOVL C02063 V=800.0 PL=0
MOVL C02064 V=800.0 PL=0
MOVL C02065 V=800.0 PL=0
MOVL C02066 V=800.0 PL=0
MOVL C02067 V=800.0 PL=0
MOVL C02068 V=800.0 PL=0
MOVL C02069 V=800.0 PL=0
MOVL C02070 V=800.0 PL=0
MOVL C02071 V=800.0 PL=0
MOVL C02072 V=800.0 PL=0
MOVL C02073 V=800.0 PL=0
MOVL C02074 V=800.0 PL=0
MOVL C02075 V=800.0 PL=0
MOVL C02076 V=800.0 PL=0
MOVL C02077 V=800.0 PL=0
MOVL C02078 V=800.0 PL=0
MOVL C02079 V=800.0 PL=0
MOVL C02080 V=800.0 PL=0
MOVL C02081 V=800.0 PL=0
MOVL C02082 V=800.0 PL=0
MOVL C02083 V=800.0 PL=0
MOVL C02084 V=800.0 PL=0
MOVL C02085 V=800.0 PL=0
MOVL C02086 V=800.0 PL=0
MOVL C02087 V=800.0 PL=0
MOVL C02088 V=800.0 PL=0
MOVL C02089 V=800.0 PL=0
MOVL C02090 V=800.0 PL=0
MOVL C02091 V=800.0 PL=0
MOVL C02092 V=800.0 PL=0
MOVL C02093 V=800.0 PL=0
MOVL C02094 V=800.0 PL=0
MOVL C02095 V=800.0 PL=0
MOVL C02096 V=800.0 PL=0
MOVL C02097 V=800.0 PL=0
MOVL C02098 V=800.0 PL=0
MOVL C02099 V=800.0 PL=0
MOVL C02100 V=800.0 PL=0
MOVL C02101 V=800.0 PL=0
MOVL C02102 V=800.0 PL=0
MOVL C02103 V=800.0 PL=0
MOVL C02104 V=800.0 PL=0
MOVL C02105 V=800.0 PL=0
MOVL C02106 V=800.0 PL=0
